IF eState = E_MethodKeepAliveMotionSystem.eIdle THEN
	MEMSET(ADR(stRtPartActivatePosition), 0, SIZEOF(stRtPartActivatePosition));
	stRtPartActivatePosition.Busy := TRUE;
	
	    nPartActivateIndex := nPartIndex;
	nPositionActivateIndex := nPositionIndex;
	  
	              eState := E_MethodKeepAliveMotionSystem.ePartActivatePosition;
	PartActivatePosition := TRUE;
ELSE
	PartActivatePosition := FALSE;
END_IF
END_METHOD

METHOD PartAllowEnable : BOOL
VAR_INPUT
	nPartID		: UDINT;
END_VAR


IF eState = E_MethodKeepAliveMotionSystem.eIdle THEN
	MEMSET(ADR(stRtPartAllowEnable), 0, SIZEOF(stRtPartAllowEnable));
	     PartToEnableAllow := nPartID;
	           eState := E_MethodKeepAliveMotionSystem.ePartAllowEnable;
	  PartAllowEnable := TRUE;
ELSE
	PartAllowEnable := FALSE;
END_IF
END_METHOD

METHOD PartForceDisable : BOOL
VAR_INPUT
	nPartID		: UDINT;
END_VAR


IF eState = E_MethodKeepAliveMotionSystem.eIdle THEN
	MEMSET(ADR(stRtPartForceDisable), 0, SIZEOF(stRtPartForceDisable));
	   PartToDisable := nPartID;
	          eState := E_MethodKeepAliveMotionSystem.ePartForceDisable;
	  PartForceDisable := TRUE;
ELSE
	PartForceDisable := FALSE;
END_IF
END_METHOD

METHOD PartForceEnable : BOOL
VAR_INPUT
	nPartID		: UDINT;
END_VAR


IF  eState  = E_MethodKeepAliveMotionSystem.eIdle
AND nPartID > 0 
THEN
		MEMSET(ADR(stRtPartForceEnable), 0, SIZEOF(stRtPartForceEnable));
		PartToEnableForce := nPartID;
				   eState := E_MethodKeepAliveMotionSystem.ePartForceEnable;
		  PartForceEnable := TRUE;
ELSE
	PartForceEnable := FALSE;
END_IF
END_METHOD

METHOD PartInitialize : BOOL
VAR_INPUT
	nPartID		: OTCID;
END_VAR



IF eState = E_MethodKeepAliveMotionSystem.eIdle THEN
	MEMSET(ADR(stRtPartInitialize), 0, SIZEOF(stRtPartInitialize));
	PartToInitialze := nPartID;
	       eState := E_MethodKeepAliveMotionSystem.ePartInitialize;
	  PartInitialize := TRUE;
ELSE
	PartInitialize := FALSE;
END_IF
END_METHOD

METHOD PartInitializeMulti : BOOL
VAR_INPUT
	
	AdrPartID		: PVOID;
	nPartCount		: UINT;
	
END_VAR

IF eState = E_MethodKeepAliveMotionSystem.eIdle THEN
	MEMSET(ADR(stRtPartInitializeMulti), 0, SIZEOF(stRtPartInitializeMulti));
	
	AddressArrayPartID	:= AdrPartID;
	          nPartCnt	:= nPartCount;		
	
	       eState := E_MethodKeepAliveMotionSystem.ePartInitializeMulti;
	  PartInitializeMulti := TRUE;
ELSE
	PartInitializeMulti := FALSE;
END_IF
END_METHOD

METHOD PartReset : BOOL
VAR_INPUT
	nPartID		: UDINT;
END_VAR


IF eState = E_MethodKeepAliveMotionSystem.eIdle THEN
	MEMSET(ADR(stRtPartReset), 0, SIZEOF(stRtPartReset));
	      PartToReset := nPartID;
	           eState := E_MethodKeepAliveMotionSystem.ePartReset;
	        PartReset := TRUE;
ELSE
	PartReset := FALSE;
END_IF
END_METHOD

METHOD RemoveEnvironmentFromGroup : BOOL
IF eState = E_MethodKeepAliveMotionSystem.eIdle THEN
	MEMSET(ADR(stRtRemoveEnvironment), 0, SIZEOF(stRtRemoveEnvironment));
	eState := E_MethodKeepAliveMotionSystem.eRemoveEnvironmentFromGroup;
	RemoveEnvironmentFromGroup := TRUE;
ELSE
	RemoveEnvironmentFromGroup := FALSE;
END_IF
END_METHOD

METHOD RemoveMoverFromGroup : BOOL
VAR_INPUT
	ipMover		: I_XPlanarMoverStandard;
END_VAR
IF eState = E_MethodKeepAliveMotionSystem.eIdle THEN
	MEMSET(ADR(stRtRemoveMover), 0, SIZEOF(stRtRemoveMover));
	eState := E_MethodKeepAliveMotionSystem.eRemoveMoverFromGroup;
	MoverToRemove := ipMover;
	RemoveMoverFromGroup := TRUE;
ELSE
	RemoveMoverFromGroup := FALSE;
END_IF
END_METHOD

METHOD RemoveMoversFromGroup : BOOL
IF eState = E_MethodKeepAliveMotionSystem.eIdle THEN
	MEMSET(ADR(stRtRemoveMovers), 0, SIZEOF(stRtRemoveMovers));
	eState := E_MethodKeepAliveMotionSystem.eRemoveMoversFromGroup;
	RemoveMoversFromGroup := TRUE;
ELSE
	RemoveMoversFromGroup := FALSE;
END_IF
END_METHOD

METHOD RemoveTracksFromGroup : BOOL



VAR_INST
	nTestCounter01 : UINT;	
	
END_VAR
IF eState = E_MethodKeepAliveMotionSystem.eIdle THEN
	MEMSET(ADR(stRtRemoveTracks), 0, SIZEOF(stRtRemoveTracks));
	eState := E_MethodKeepAliveMotionSystem.eRemoveTracksFromGroup;
	RemoveTracksFromGroup := TRUE;
	
	nTestCounter01 := nTestCounter01 +1;
ELSE
	RemoveTracksFromGroup := FALSE;
END_IF
END_METHOD

METHOD ResetGroup : BOOL
IF eState = E_MethodKeepAliveMotionSystem.eIdle THEN
	MEMSET(ADR(stRtResetGroup), 0, SIZEOF(stRtResetGroup));
	eState := E_MethodKeepAliveMotionSystem.eResetGroup;
	ResetGroup := TRUE;
ELSE
	ResetGroup := FALSE;
END_IF
END_METHOD

METHOD ResetMovers : BOOL
IF eState = E_MethodKeepAliveMotionSystem.eIdle THEN
	MEMSET(ADR(stRtResetMovers), 0, SIZEOF(stRtResetMovers));
	eState := E_MethodKeepAliveMotionSystem.eResetMovers;
	ResetMovers := TRUE;
ELSE
	ResetMovers := FALSE;
END_IF
END_METHOD

METHOD ResetParts : BOOL
IF eState = E_MethodKeepAliveMotionSystem.eIdle THEN
	MEMSET(ADR(stRtResetParts), 0, SIZEOF(stRtResetParts));
	eState := E_MethodKeepAliveMotionSystem.eResetParts;
	ResetParts := TRUE;
ELSE
	ResetParts := FALSE;
END_IF
END_METHOD

METHOD ResetTracks : BOOL
IF eState = E_MethodKeepAliveMotionSystem.eIdle THEN
	MEMSET(ADR(stRtResetTracks), 0, SIZEOF(stRtResetTracks));
	eState := E_MethodKeepAliveMotionSystem.eResetTracks;
	ResetTracks := TRUE;
ELSE
	ResetTracks := FALSE;
END_IF
END_METHOD

METHOD UtilityCheckForError : DINT
VAR_INPUT
	bAutoReset : BOOL;
END_VAR
	IF bAutoReset THEN
		IF ipXpuInternal.Error THEN
			ipXpuInternal.ErrorAcknowledge();
		END_IF
	END_IF

	IF ipXpuInternal.Error THEN
		UtilityCheckForError := -1;
	ELSE
		UtilityCheckForError := +1;
	END_IF
END_METHOD

METHOD UtilityErrorReset : BOOL
VAR_INPUT
END_VAR
IF ipXpuInternal.Error THEN
	ipXpuInternal.ErrorAcknowledge();
END_IF
END_METHOD

METHOD PROTECTED ccl_AddEnvironmentToGroup : BOOL

VAR
	EmptyOT : EPlanarObjectType;
END_VAR

CASE nState OF
	

	0:  // Prepare
		stRtAddEnvironment.Aborted := FALSE;
		stRtAddEnvironment.Active  := TRUE;
		stRtAddEnvironment.Done    := FALSE;
		stRtAddEnvironment.Busy    := TRUE;
		stRtAddEnvironment.Error   := FALSE;
		stRtAddEnvironment.ErrorID := 0;
		stRtAddEnvironment.stInfo  := _stResultErrorInfoClear;
		
		nState := 5;


	5:  // Checking if the environment already belongs to the group
		IF environment.MCTOPLC_STD.GroupOID = 0 THEN
			environment.CreateBoundary(cmdFeedback);
			nState := 10;
		ELSE
			nState := 110;
		END_IF
	
		
	10:	// Creating the boundary 
		environment.CreateBoundary(cmdFeedback);
		nState := nState + 1;
			
	11:	IF cmdFeedback.Done THEN
			nState := 20;
		ELSIF cmdFeedback.Error THEN
			nState := 100;
		END_IF
		
		
	20:	// Adding the environment to the group
		environment.AddToGroup(cmdFeedback, group);
		nState := nState + 1;

	21:	IF cmdFeedback.Done 
		OR cmdFeedback.Error
		THEN
			nState := 100;
		END_IF
		
		
		
	100: // Result with action
		stRtAddEnvironment.Aborted            := FALSE;
		stRtAddEnvironment.Active             := FALSE;
		stRtAddEnvironment.Busy               := FALSE;
		stRtAddEnvironment.Done               := cmdFeedback.Done;
		stRtAddEnvironment.Error              := cmdFeedback.Error;
		stRtAddEnvironment.ErrorID            := cmdFeedback.ErrorId;
		stRtAddEnvironment.stInfo.nObjectID   := cmdFeedback.objectInfo.Id;
		stRtAddEnvironment.stInfo.nObjectType := cmdFeedback.objectInfo.ObjectType;
		nState := 200;
		
		
	110: // Result without action
		stRtAddEnvironment.Aborted            := FALSE;
		stRtAddEnvironment.Active             := FALSE;
		stRtAddEnvironment.Busy               := FALSE;
		stRtAddEnvironment.Done               := TRUE;
		stRtAddEnvironment.Error              := FALSE;
		stRtAddEnvironment.ErrorID            := 0;
		stRtAddEnvironment.stInfo.nObjectID   := 0;
		stRtAddEnvironment.stInfo.nObjectType := EmptyOT;
		nState := 200;		
		
		
	200: // Done	
		eState := E_MethodKeepAliveMotionSystem.eIdle;
		nState := 0;		
		ccl_AddEnvironmentToGroup := TRUE;
		
		
END_CASE
END_METHOD

METHOD PROTECTED ccl_AddModuleToEnvironment : BOOL

CASE nState OF
	
	0: 	// Prepare
		stRtAddModule.Aborted := FALSE;
		stRtAddModule.Active  := TRUE;
		stRtAddModule.Busy	  := TRUE;
		stRtAddModule.Done 	  := FALSE;
		stRtAddModule.Error   := FALSE;
		stRtAddModule.ErrorID := 0;
		stRtAddModule.stInfo  := _stResultErrorInfoClear;
		nState := 10;
	
		
	10: // Adding the tile	
		environment.AddStator(cmdFeedback, _addModulePositionX, _addModulePositionY);
		nState := nState + 10;
		
		
	20: // Checking command feedback
		IF cmdFeedback.Done
		OR cmdFeedback.Error
		THEN
			                  _bResultDone  := cmdFeedback.Done;
			                  _bResultError := cmdFeedback.Error;
			                _nResultErrorID := cmdFeedback.ErrorId;
			   _stResultErrorInfo.nObjectID := cmdFeedback.objectInfo.Id;	
			 _stResultErrorInfo.nObjectType := cmdFeedback.objectInfo.ObjectType;	
			    		 nState := 100;
		END_IF		

		
	100:  // Done	
		stRtAddModule.Aborted	:= FALSE;
		stRtAddModule.Active	:= FALSE;
		stRtAddModule.Busy   	:= FALSE;
		stRtAddModule.Done   	:= _bResultDone;
		stRtAddModule.Error		:= _bResultError;
		stRtAddModule.ErrorID	:= _nResultErrorID;
		stRtAddModule.stInfo	:= _stResultErrorInfo;
		
		eState := E_MethodKeepAliveMotionSystem.eIdle;
		nState := 0;
		ccl_AddModuleToEnvironment := TRUE;	

END_CASE
END_METHOD

METHOD PROTECTED ccl_AddMoversToGroup : BOOL



CASE nState OF
	
	0:  // Prepare
		stRtAddMovers.Aborted := FALSE;
		stRtAddMovers.Active  := FALSE;
		stRtAddMovers.Busy    := TRUE;
		stRtAddMovers.Error   := FALSE;
		stRtAddMovers.ErrorID := 0;
		stRtAddMovers.stInfo  := _stResultErrorInfoClear;

		nState := 10;
	
	
	10: // Adding movers to the group
		stRtAddMovers.Active := TRUE;
		bDone := TRUE;
		FOR nForCounter := 1 TO _nAxisCount DO
			IF ipMover[nForCounter].P_PhysicalAreaID > 0 THEN
				bDone := bDone AND ipMover[nForCounter].AddToGroup(group);
			END_IF
		END_FOR
		IF bDone THEN
			nState := 20;
		END_IF
		
		
	20: // Checking command feedback
		_nResultErrorID    := 0;
		_stResultErrorInfo := _stResultErrorInfoClear;
	
		bError := FALSE;
		bDone  := TRUE;
		FOR nForCounter := 1 TO _nAxisCount DO
			IF ipMover[nForCounter].P_PhysicalAreaID > 0 THEN	
				bDone := bDone  AND ipMover[nForCounter].P_AddToGroup.Done;
				
				IF ipMover[nForCounter].P_AddToGroup.Error THEN
						bError := TRUE;
					   _nResultErrorID := ipMover[nForCounter].P_AddToGroup.ErrorID;
					_stResultErrorInfo := ipMover[nForCounter].P_AddToGroup.stInfo;
				END_IF
			END_IF
		END_FOR
		
		IF bDone 
		OR bError
		THEN
			_bResultDone  := bDone;
			_bResultError := bError;	
				   nState := 100;		
		END_IF
		
		
	100:  // Done
		stRtAddMovers.Aborted 	:= FALSE;
		stRtAddMovers.Active	:= FALSE;
		stRtAddMovers.Busy	    := FALSE;
		stRtAddMovers.Done      := _bResultDone;
		stRtAddMovers.Error     := _bResultError;
		stRtAddMovers.ErrorID	:= _nResultErrorID;
		stRtAddMovers.stInfo    := _stResultErrorInfo;
		
		eState := E_MethodKeepAliveMotionSystem.eIdle;
		nState := 0;
		ccl_AddMoversToGroup := TRUE;
		

END_CASE
END_METHOD

METHOD PROTECTED ccl_AddMoverToGroup : BOOL


VAR_INPUT
	ipMoverToAdd	: I_XPlanarMoverStandard;
END_VAR


VAR_INST
	nMoverToAdd		: UDINT;	
END_VAR


CASE nState OF

	0: // Prepare
		stRtAddMover.Aborted := FALSE;
		stRtAddMover.Active  := TRUE;
		stRtAddMover.Busy    := TRUE;
		stRtAddMover.Done    := FALSE;
		stRtAddMover.Error	 := FALSE;
		stRtAddMover.ErrorID := 0;
		stRtAddMover.stInfo	 := _stResultErrorInfoClear;
		
		nState := 10;
	
	10: // Adding the mover to the group
		      bDone := TRUE;		
		nMoverToAdd := 0;
		FOR idx:=1 TO Params_XPlanar.maxNumMover DO
			IF  ipMover[idx] <> 0			 
			AND ipMover[idx] = ipMoverToAdd
			THEN
				nMoverToAdd := idx;	
				EXIT;
			END_IF
		END_FOR
		
		IF nMoverToAdd > 0 THEN
			ipMover[nMoverToAdd].AddToGroup(group);
			nState := 20;	
		ELSE
			nState := 30;	
		END_IF
		

	20: // Checking feedback
		_bResultDone       := ipMover[nMoverToAdd].P_AddToGroup.Done;
		_bResultError      := ipMover[nMoverToAdd].P_AddToGroup.Error;
		_nResultErrorID    := ipMover[nMoverToAdd].P_AddToGroup.ErrorID;
		_stResultErrorInfo := ipMover[nMoverToAdd].P_AddToGroup.stInfo;
		
		IF _bResultDone
		OR _bResultError
		THEN
			nState := 100;
		END_IF
		
		
	30:	// Error - no mover to add = undefined error
		_bResultDone       := FALSE;
		_bResultError      := TRUE;
		_nResultErrorID    := 0;
		_stResultErrorInfo := _stResultErrorInfoClear;		
		            nState := 100;
	
		
	100: // Done	
		stRtAddMover.Active  := FALSE;		
		stRtAddMover.Busy    := FALSE;
		stRtAddMover.Done    := _bResultDone;		
		stRtAddMover.Error   := _bResultError;
		stRtAddMover.ErrorID := _nResultErrorID;
		stRtAddMover.stInfo  := _stResultErrorInfo; 			

		eState := E_MethodKeepAliveMotionSystem.eIdle;
		nState := 0;		
		ccl_AddMoverToGroup := TRUE;
		

END_CASE
END_METHOD

METHOD PROTECTED ccl_AddTracksToGroup : BOOL



VAR_INST
	
	nTestCounter01	: UINT;
	
END_VAR
CASE nState OF
	
	0:  // Prepare
		stRtAddTracks.Aborted  := FALSE;
		stRtAddTracks.Active   := TRUE;
		stRtAddTracks.Busy     := TRUE;
		stRtAddTracks.Done     := FALSE;
		stRtAddTracks.Error    := FALSE;
		stRtAddTracks.ErrorID  := 0;
		stRtAddTracks.stInfo   := _stResultErrorInfoClear;

		nState := 10;
		
		nTestCounter01 := nTestCounter01 +1;
	
		
	10: // Adding tracks to the group
		bDone := TRUE;
		FOR nForCounter := 1 TO _nTrackCount DO
			bDone := bDone AND ipTrack[nForCounter].AddToGroup(group);
		END_FOR
		
		IF bDone THEN
			nState := 20;
		END_IF
		
		
	20: // Checking feedback 
		nErrorID := 0;
		  bError := FALSE;
		   bDone := TRUE;
		   
		FOR nForCounter := 1 TO _nTrackCount DO
			 bDone := bDone  AND ipTrack[nForCounter].P_AddToGroup.Done;
		
			IF NOT bError AND ipTrack[nForCounter].P_AddToGroup.Error THEN
				           bError := TRUE;
				         nErrorID := ipTrack[nForCounter].P_AddToGroup.ErrorID;
				stResultErrorInfo := ipTrack[nForCounter].P_AddToGroup.stInfo;
			END_IF
		END_FOR
		
		IF bDone OR bError THEN
			      _bResultDone := bDone;
			     _bResultError := bError;
			   _nResultErrorID := nErrorID;
			_stResultErrorInfo := stResultErrorInfo;
			            nState := 100;
		END_IF
		
	
	100:  // Done
		stRtAddTracks.Active  := FALSE;
		stRtAddTracks.Busy    := FALSE;
		stRtAddTracks.Done    := _bResultDone;
		stRtAddTracks.Error   := _bResultError;
		stRtAddTracks.ErrorID := _nResultErrorID;
		stRtAddTracks.stInfo  := _stResultErrorInfo;
		
		eState := E_MethodKeepAliveMotionSystem.eIdle;
		nState := 0;			   
		ccl_AddTracksToGroup  := TRUE;

END_CASE
END_METHOD

METHOD ccl_CheckValidMovers : BOOL
VAR_INPUT
END_VAR



VAR_INST
	
	nState		 : UDINT;
	
	nHardwareOID				: UDINT;
	nModuleOID					: UDINT;
	nParameterOID				: UDINT;
	nSizeOfParameter			: UDINT;
	ParameterAddress			: PVOID;
	
	
	fbReadReq    : ADSREAD := ( NETID := '', PORT := 501, TMOUT := DEFAULT_ADS_TIMEOUT );
	bReadADS	 : BOOL;	
	bReadBusy	 : BOOL;
	bReadError	 : BOOL;
	nReaderrorID : UDINT;
	
	
	ModuleOIDs		: ARRAY[1..Param_TcIoXPlanarEnvironment.MaxXPlanarMoversPerXpu] OF OTCID;
	nMoverIdx		: UINT;
	
	
	//PROPERTY ipTcIoMover : ARRAY [1..Params_XPlanar.maxNumMover] OF I_TcIoXPlanarMover;
	
	Movers					: ARRAY [1..Params_XPlanar.maxNumMover] OF I_TcIoXPlanarMover;
	MoverPositionInfoAct	: MoverPositionInfo;
	
	
	nMoverValidCount		: UDINT;	
	bAllMoversValid			: BOOL;
	bMoverLost				: BOOL;

	
	fCurrentPositionX_01		: LREAL;
	fCurrentPositionX_02		: LREAL;
	fFeedbackCheckRegister		: ARRAY [0..10] OF LREAL;
	nFeedbackCheckIdx			: UINT;
	idx							: UINT;
	nMatchCount					: UINT;
	bFreezeDetect				: BOOL;
	
	
END_VAR


	CASE nState OF
		
	0:	
		stValidMoverCheckInfo.bDone            := FALSE;
		stValidMoverCheckInfo.bAllMoversValid  := FALSE;
		stValidMoverCheckInfo.bMoverLost       := FALSE;
		stValidMoverCheckInfo.nValidMoverCount := 0;
	
		       nMoverIdx := 0;
			  bMoverLost := FALSE;
		nMoverValidCount := 0;
		          nState := 10;
				  
	10:
		nMoverIdx := nMoverIdx +1;
		IF nMoverIdx <= Params_XPlanar.maxNumMover AND nMoverIdx <= ipXpuInternal.GetMoverCount() AND ipMover[nMoverIdx] <> 0 THEN
			nState := nState + 10;
		ELSE
			nMoverIdx := nMoverIdx -1;
			   nState := 30;
		END_IF
	
	20:		
		IF ipMover[nMoverIdx] <> 0 AND nMoverIdx <= ipXpuInternal.GetMoverCount() THEN
			MoverPositionInfoAct := ipXpuInternal.MoverTcIo(nMoverIdx).GetActualPositions();
			IF  MoverPositionInfoAct.MovementAreaOID  <> 0
			AND MoverPositionInfoAct.ActualPosition.z  < 6.0
			THEN
				nMoverValidCount := nMoverValidCount +1;
			END_IF
			nState := nState - 10;
		END_IF

	30:
		IF nMoverValidCount = nMoverIdx THEN 
			bAllMoversValid := TRUE;
			nState := nState + 10; 
		ELSE
			bMoverLost := TRUE;
			nState := 100;
		END_IF
		
				
		
	40: // Check Feedback
		  nMoverIdx := 0;
		nMatchCount := 0;
		nState := nState + 1; 
		
	41:
		nMoverIdx := nMoverIdx +1;
		IF nMoverIdx <= Params_XPlanar.maxNumMover AND nMoverIdx <= ipXpuInternal.GetMoverCount() AND ipMover[nMoverIdx] <> 0 THEN
			nState := nState + 1; 
		ELSE
			nState := 100;
		END_IF
	

	42:
		MoverPositionInfoAct := ipXpuInternal.MoverTcIo(nMoverIdx).GetActualPositions();		
		fCurrentPositionX_01 := MoverPositionInfoAct.ActualPosition.x; 
		nState := nState + 1; 
		
	43:
		MoverPositionInfoAct := ipXpuInternal.MoverTcIo(nMoverIdx).GetActualPositions();		
		fCurrentPositionX_02 := MoverPositionInfoAct.ActualPosition.x;
		
		IF fCurrentPositionX_01 = fCurrentPositionX_02 THEN
			nMatchCount := nMatchCount +1;
			
			IF nMatchCount >= 4 THEN
				bFreezeDetect := TRUE;
				nState := nState + 1; 
			ELSE
				nState := nState - 1; 
			END_IF
		ELSE
			bFreezeDetect := FALSE;
			nState := nState + 1; 
		END_IF
		
	44:
		IF bFreezeDetect THEN
			bAllMoversValid := FALSE;
			     bMoverLost := TRUE;
	       nMoverValidCount := 0;
				 
			nState := 100;
		ELSE
			nState := 41;
		END_IF


		
		
	
	100:		
		stValidMoverCheckInfo.bAllMoversValid 	:= bAllMoversValid;
		stValidMoverCheckInfo.bMoverLost 		:= bMoverLost; 
		stValidMoverCheckInfo.bDone 			:= TRUE;
		stValidMoverCheckInfo.nValidMoverCount  := nMoverValidCount;
	
		eState := E_MethodKeepAliveMotionSystem.eIdle;
		nState := 0;
		
		
	
	END_CASE
END_METHOD

METHOD PROTECTED ccl_DisableGroup : BOOL

CASE nState OF 


	0:  // Prepare 
		stRtDisableGroup.Aborted  := FALSE;
		stRtDisableGroup.Active   := TRUE;
		stRtDisableGroup.Busy     := TRUE;
		stRtDisableGroup.Done     := FALSE;
		stRtDisableGroup.Error    := FALSE;
		stRtDisableGroup.ErrorID  := 0;
		stRtDisableGroup.stInfo   := _stResultErrorInfoClear;
	
		nState := 10;


	10: // Disabeling the group
		Group.Disable(CmdFeedback);
		nState := 20; 
		
		
	20: // Checking feedback
		                  _bResultDone := CmdFeedback.Done;
		                 _bResultError := CmdFeedback.Error;
		               _nResultErrorID := CmdFeedback.ErrorId;
		  _stResultErrorInfo.nObjectID := CmdFeedback.objectInfo.Id;   
		_stResultErrorInfo.nObjectType := CmdFeedback.objectInfo.ObjectType;
	
		IF _bResultDone
		OR _bResultError
		THEN
			nState := 100;	
		END_IF
	
		
	100:  // Done
		stRtDisableGroup.Aborted := FALSE;
		stRtDisableGroup.Active  := FALSE;
		stRtDisableGroup.Busy    := FALSE;
		stRtDisableGroup.Done    := _bResultDone;
		stRtDisableGroup.Error	 := _bResultError;
		stRtDisableGroup.ErrorID := _nResultErrorID;
		stRtDisableGroup.stInfo  := _stResultErrorInfo;
	
		eState := E_MethodKeepAliveMotionSystem.eIdle;
		nState := 0;	
		ccl_DisableGroup := TRUE;
			
END_CASE
END_METHOD

METHOD PROTECTED ccl_DisableMovers : BOOL



CASE nState OF
	

	0:  // Prepare
		stRtDisableMovers.Aborted  := FALSE;
		stRtDisableMovers.Active   := TRUE;
		stRtDisableMovers.Busy     := TRUE;
		stRtDisableMovers.Done	   := FALSE;
		stRtDisableMovers.Error    := FALSE;
		stRtDisableMovers.ErrorID  := 0;
		stRtDisableMovers.stInfo   := _stResultErrorInfoClear;
	
		nErrorID := 0;
		nState:= 10;
	
		
	10: // Disable all movers
		FOR nForCounter := 1 TO _nAxisCount DO
			IF ipMover[nForCounter].P_PhysicalAreaID > 0 THEN
				ipMover[nForCounter].Disable('Disable all Movers');
			END_IF
		END_FOR
		nState := 20;
		
		
	20:  // Checking feedback
		 bDone := TRUE;
		bError := FALSE;
		FOR nForCounter := 1 TO _nAxisCount DO
			IF ipMover[nForCounter].P_PhysicalAreaID > 0 THEN
				bDone := bDone AND ipMover[nForCounter].P_Disable.Done;
				
				IF NOT bError AND ipMover[nForCounter].P_Disable.Error THEN
							   bError := TRUE;
							 nErrorID := ipMover[nForCounter].P_Disable.ErrorID;
					stResultErrorInfo := ipMover[nForCounter].P_Disable.stInfo;
				END_IF
			END_IF
		END_FOR	
			
		IF bDone OR bError THEN
			nState := 21;
		END_IF

	21:
		_bResultDone 		:= bDone;
		_bResultError 		:= bError;
		_nResultErrorID		:= nErrorID;
		_stResultErrorInfo	:= stResultErrorInfo;
		nState := 100;
		
	
	100:  // Done
		stRtDisableMovers.Aborted  := FALSE;
		stRtDisableMovers.Active   := FALSE;
		stRtDisableMovers.Busy     := FALSE;
		stRtDisableMovers.Done	   := _bResultDone;
		stRtDisableMovers.Error    := _bResultError;
		stRtDisableMovers.ErrorID  := _nResultErrorID;
		stRtDisableMovers.stInfo   := _stResultErrorInfo;		
	
		eState := E_MethodKeepAliveMotionSystem.eIdle;
		nState := 0;
		ccl_DisableMovers := TRUE;
		
END_CASE
END_METHOD

METHOD PROTECTED ccl_DisableTracks : BOOL

VAR_INST

	nTrackToDisable		: INT;
	nTrackToDisableCNT	: INT;
		
	nTestCounter01		: UINT;
	nTestCounter02		: UINT;
	nLastTrackDisabled 	: INT;
	
END_VAR
CASE nState OF
	

	0:  // Prepare
		stRtDisableTracks.Aborted  := FALSE;
		stRtDisableTracks.Active   := TRUE;
		stRtDisableTracks.Busy     := TRUE;
		stRtDisableTracks.Done     := FALSE; 
		stRtDisableTracks.Error    := FALSE; 
		stRtDisableTracks.ErrorID  := 0;
		stRtDisableTracks.stInfo   := _stResultErrorInfoClear;
	
		nState := 10;
		
		nTestCounter01 := nTestCounter01 +1;
		
		
	10:  // Disabeling all tracks one-by-one
			     nTestCounter02 := nTestCounter02 +1;
				 
				 		  bError := FALSE;
				           bDone := FALSE;
		         nTrackToDisable := 0;
		      nTrackToDisableCNT := 0;
	          nLastTrackDisabled := 0;
		stRtEnableTracks.Active := TRUE;
		                 nState := 11;
		
	11:	// Checking if track is real
		nTrackToDisableCNT := nTrackToDisableCNT +1;
		IF nTrackToDisableCNT <= _nTrackCount THEN
			IF ipTrack[nTrackToDisableCNT] <> 0 THEN
				   nTrackToDisable := nTrackToDisableCNT;
				nLastTrackDisabled := nTrackToDisable;
				nState := nState +1;
			ELSE
				nState := 20;
			END_IF
		ELSE
			 bDone := TRUE;
			nState := 20;
		END_IF
		
		
	12:	// Disabeling
		IF ipTrack[nTrackToDisable].Disable() THEN
			nState := nState +1;
		END_IF
	
			
	13:	// Checking feedback
		IF ipTrack[nTrackToDisable].P_Disable.Done THEN
			nState := nState -2;
		ELSIF ipTrack[nTrackToDisable].P_Disable.Error THEN
				         bError := ipTrack[nTrackToDisable].P_Disable.Error;
				       nErrorID := ipTrack[nTrackToDisable].P_Disable.ErrorID;
			  stResultErrorInfo := ipTrack[nTrackToDisable].P_Disable.stInfo;
		
			nState := 20;
		END_IF
			
	
	20:	// All tracks are through
				  _bResultDone := bDone;
				 _bResultError := bError;
			   _nResultErrorID := nErrorID;
			_stResultErrorInfo := stResultErrorInfo;		

			nState := 100;				
	
	
	100:  // Done	
		stRtDisableTracks.Active   := FALSE;
		stRtDisableTracks.Busy     := FALSE;
		stRtDisableTracks.Done 	   := _bResultDone;
		stRtDisableTracks.Error    := _bResultError;
		stRtDisableTracks.ErrorID  := _nResultErrorID;
		stRtDisableTracks.stInfo   := _stResultErrorInfo;
		
		           eState := E_MethodKeepAliveMotionSystem.eIdle;
				   nState := 0;
		ccl_DisableTracks := TRUE;
		
			
END_CASE
END_METHOD

METHOD PROTECTED ccl_EnableGroup : BOOL




CASE nState OF 
	
	0:  // Prepare
		stRtEnableGroup.Aborted  := FALSE;
		stRtEnableGroup.Active   := TRUE;
		stRtEnableGroup.Busy     := TRUE;
		stRtEnableGroup.Done     := FALSE;
		stRtEnableGroup.Error    := FALSE;
		stRtEnableGroup.ErrorID  := 0;
		stRtEnableGroup.stInfo   := _stResultErrorInfoClear;
	
		nState := 10;
	
	
	10: // Activating the group
		group.Enable(cmdFeedback);
		nState := 11;
	
	
	11: // Checking feedback
		                  _bResultDone := cmdFeedback.Done;
		                 _bResultError := cmdFeedback.Error;
		               _nResultErrorID := cmdFeedback.ErrorId;
		  _stResultErrorInfo.nObjectID := cmdFeedback.objectInfo.Id;
		_stResultErrorInfo.nObjectType := cmdFeedback.objectInfo.ObjectType;
	
		IF _bResultDone OR _bResultError THEN
			nState := 100;
		END_IF
	
		
	100:  // Done
		stRtEnableGroup.Aborted  := FALSE;
		stRtEnableGroup.Active   := FALSE;
		stRtEnableGroup.Busy     := FALSE;
		stRtEnableGroup.Done     := _bResultDone;
		stRtEnableGroup.Error    := _bResultError;
		stRtEnableGroup.ErrorID  := _nResultErrorID;
		stRtEnableGroup.stInfo   := _stResultErrorInfo;	
	
		eState := E_MethodKeepAliveMotionSystem.eIdle;
		nState := 0;
		ccl_EnableGroup := TRUE;
	
		
END_CASE
END_METHOD

METHOD PROTECTED ccl_EnableMovers : BOOL


CASE nState OF

	0:	// Prepare 
		stRtEnableMovers.Aborted  := FALSE;
		stRtEnableMovers.Active   := TRUE;
		stRtEnableMovers.Busy	  := TRUE;
		stRtEnableMovers.Done     := FALSE;
		stRtEnableMovers.Error    := FALSE;
		stRtEnableMovers.ErrorID  := 0;
		stRtEnableMovers.stInfo	  := _stResultErrorInfoClear;

		nState := 10;
		
		
	10:  // Enabeling all movers
		bDone := TRUE;
		FOR nForCounter := 1 TO _nAxisCount DO
			IF ipMover[nForCounter].P_PhysicalAreaID > 0 THEN
				bDone := bDone AND ipMover[nForCounter].Enable('Enable all Movers');
			END_IF
		END_FOR
		IF bDone THEN
			nState := 20;
		END_IF
		
	20:  // Checking feedback
		 bDone := TRUE;
		bError := FALSE;
		FOR nForCounter := 1 TO _nAxisCount DO
			IF ipMover[nForCounter].P_PhysicalAreaID > 0 THEN
				bDone := bDone AND ipMover[nForCounter].P_Enable.Done;
			
				IF NOT bError AND ipMover[nForCounter].P_Enable.Error THEN
							   bError := TRUE;
							 nErrorID := ipMover[nForCounter].P_Enable.ErrorID;
					stResultErrorInfo := ipMover[nForCounter].P_Enable.stInfo;
				END_IF	
			END_IF
		END_FOR	
		
		IF bDone OR bError THEN
				  _bResultDone := bDone;
				 _bResultError := bError;
			   _nResultErrorID := nErrorID;
			_stResultErrorInfo := stResultErrorInfo;			
		
			nState := 100;
		END_IF
		
			
	100:  // Done
		stRtEnableMovers.Aborted  := FALSE;
		stRtEnableMovers.Active   := FALSE;
		stRtEnableMovers.Busy	  := FALSE;
		stRtEnableMovers.Done     := _bResultDone;
		stRtEnableMovers.Error    := _bResultError;
		stRtEnableMovers.ErrorID  := _nResultErrorID;
		stRtEnableMovers.stInfo	  := _stResultErrorInfo;
	
		eState := E_MethodKeepAliveMotionSystem.eIdle;
		nState := 0;
		ccl_EnableMovers := TRUE;
			

	
END_CASE
END_METHOD

METHOD PROTECTED ccl_EnableTrack : BOOL

VAR_INPUT
	ipTrackToEnable	: I_TrackStandard;
END_VAR






CASE nState OF

	0:  // Prepare
		stRtEnableTrack.Aborted := FALSE;
		stRtEnableTrack.Active  := TRUE;
		stRtEnableTrack.Busy    := TRUE;
		stRtEnableTrack.Done    := FALSE;
		stRtEnableTrack.Error   := FALSE;
		stRtEnableTrack.ErrorID := 0;
		stRtEnableTrack.stInfo  := _stResultErrorInfoClear;

		nState := 10;
		
		
	10: // Enable the track
		IF ipTrackToEnable.Enable() THEN
			nState := 20;
		END_IF
	
	
	20: // Checking feedback
		 _bResultDone := ipTrackToEnable.P_Enable.Done;
		_bResultError := ipTrackToEnable.P_Enable.Error;		
	
		IF _bResultDone OR _bResultError THEN
			        _nResultErrorID := ipTrackToEnable.P_Enable.ErrorID;
			     _stResultErrorInfo := ipTrackToEnable.P_Enable.stInfo;
			nState := 100;
		END_IF
		

	100: // Done
		stRtEnableTrack.Aborted := FALSE;
		stRtEnableTrack.Active  := FALSE;
		stRtEnableTrack.Busy    := FALSE;
		stRtEnableTrack.Done    := _bResultDone;
		stRtEnableTrack.Error   := _bResultError;
		stRtEnableTrack.ErrorID := _nResultErrorID;
		stRtEnableTrack.stInfo  := _stResultErrorInfo;

		         eState := E_MethodKeepAliveMotionSystem.eIdle;
				 nState := 0;
		ccl_EnableTrack := TRUE;
		
				
END_CASE
END_METHOD

METHOD PROTECTED ccl_EnableTracks : BOOL

VAR_INST

	nTrackToEnable		: INT;
	nTrackToEnableCNT	: INT;
		
	nTestCounter01		: UINT;
	nTestCounter02		: UINT;
	nLastTrackEnabled 	: INT;
	
END_VAR
CASE nState OF
	

	0:  // Prepare
		stRtEnableTracks.Aborted  := FALSE;
		stRtEnableTracks.Active   := TRUE;
		stRtEnableTracks.Busy     := TRUE;
		stRtEnableTracks.Done     := FALSE; 
		stRtEnableTracks.Error    := FALSE; 
		stRtEnableTracks.ErrorID  := 0;
		stRtEnableTracks.stInfo   := _stResultErrorInfoClear;
	
		nState := 10;
		
		nTestCounter01 := nTestCounter01 +1;
		
		
	10:  // Enabeling all tracks one-by-one
			     nTestCounter02 := nTestCounter02 +1;
				 
				 		 bError := FALSE;
				          bDone := FALSE;
		         nTrackToEnable := 0;
		      nTrackToEnableCNT := 0;
	          nLastTrackEnabled := 0;
		stRtEnableTracks.Active := TRUE;
		                 nState := 11;
		
	11:	// Checking if track is real
		nTrackToEnableCNT := nTrackToEnableCNT +1;
		IF nTrackToEnableCNT <= _nTrackCount THEN
			IF ipTrack[nTrackToEnableCNT] <> 0 THEN
				IF ipTrack[nTrackToEnableCNT].GetLength() > 0 THEN
					   nTrackToEnable := nTrackToEnableCNT;
					nLastTrackEnabled := nTrackToEnable;
					nState := nState +1;
				END_IF
			END_IF
		ELSE
			 bDone := TRUE;
			nState := 20;
		END_IF
		
		
	12:	// Enabeling
		IF ipTrack[nTrackToEnable].Enable() THEN
			nState := nState +1;
		END_IF
	
			
	13:	// Checking feedback
		IF ipTrack[nTrackToEnable].P_Enable.Done THEN
			nState := nState -2;
		ELSIF ipTrack[nTrackToEnable].P_Enable.Error THEN
				         bError := ipTrack[nTrackToEnable].P_Enable.Error;
				       nErrorID := ipTrack[nTrackToEnable].P_Enable.ErrorID;
			  stResultErrorInfo := ipTrack[nTrackToEnable].P_Enable.stInfo;
		
			nState := 20;
		END_IF
			
	
	20:	// All tracks are through
				  _bResultDone := bDone;
				 _bResultError := bError;
			   _nResultErrorID := nErrorID;
			_stResultErrorInfo := stResultErrorInfo;		

			nState := 100;				
	
	
	100:  // Done	
		stRtEnableTracks.Active   := FALSE;
		stRtEnableTracks.Busy     := FALSE;
		stRtEnableTracks.Done 	  := _bResultDone;
		stRtEnableTracks.Error 	  := _bResultError;
		stRtEnableTracks.ErrorID  := _nResultErrorID;
		stRtEnableTracks.stInfo   := _stResultErrorInfo;
		
		          eState := E_MethodKeepAliveMotionSystem.eIdle;
				  nState := 0;
		ccl_EnableTracks := TRUE;
		
			
END_CASE
END_METHOD

METHOD PROTECTED ccl_HaltSystem : BOOL

CASE nState OF
	
	0:  // Prepare 
		stRtHaltSystem.Aborted := FALSE;
		stRtHaltSystem.Active  := TRUE;
		stRtHaltSystem.Busy    := TRUE;
		stRtHaltSystem.Done    := FALSE;
		stRtHaltSystem.Error   := FALSE;
		stRtHaltSystem.ErrorID := 0;
		stRtHaltSystem.stInfo  := _stResultErrorInfoClear;

		nState := 10;
	
		
	10: // Halt to all moving movers
		bDone := TRUE;
		FOR nForCounter := 1 TO _nAxisCount DO
			IF ipMover[nForCounter] <> 0 THEN
				IF ipMover[nForCounter].P_Busy THEN
					bDone := bDone AND ipMover[nForCounter].Halt('HaltSystem');
				ELSE
					bDone := bDone AND TRUE;
				END_IF
			END_IF 
		END_FOR
		IF bDone THEN
			nState := 20;
		END_IF
		
		
	20:  // Checking feedback
		bError := FALSE;
		  bDone:= TRUE;
		FOR nForCounter := 1 TO _nAxisCount DO
			IF ipMover[nForCounter] <> 0 THEN
				
				bDone := bDone AND (ipMover[nForCounter].P_Halt.Done OR NOT ipMover[nForCounter].P_Busy);
				
				IF NOT bError AND ipMover[nForCounter].P_Halt.Error THEN
					IF ipMover[nForCounter].P_Busy THEN	
						         nErrorID := ipMover[nForCounter].P_Halt.ErrorID;
						stResultErrorInfo := ipMover[nForCounter].P_Halt.stInfo;
						           bError := TRUE;
					END_IF 
				END_IF
				
			END_IF 
		END_FOR
		
		IF bDone OR bError THEN
				  _bResultDone := bDone;
				 _bResultError := bError;
			   _nResultErrorID := nErrorID;
			_stResultErrorInfo := stResultErrorInfo;					
		
			nState := 100;
		END_IF
		
		
	100:  // Done
		stRtHaltSystem.Aborted := FALSE;
		stRtHaltSystem.Active  := FALSE;
		stRtHaltSystem.Busy    := FALSE;
		stRtHaltSystem.Done    := _bResultDone;
		stRtHaltSystem.Error   := _bResultError;
		stRtHaltSystem.ErrorID := _nResultErrorID;
		stRtHaltSystem.stInfo  := _stResultErrorInfo;
	
		eState := E_MethodKeepAliveMotionSystem.eIdle;
		nState := 0;
		ccl_HaltSystem := TRUE;
		

	
END_CASE
END_METHOD

METHOD PROTECTED ccl_LeaveTrack : BOOL

VAR_INST
	ActPosition		: PositionXYC;
	stOptions 		: ST_LeaveTrackOptions;

END_VAR


CASE nState OF
	
	0:  // Prepare
		stRtLeaveTrack.Aborted  := FALSE;
		stRtLeaveTrack.Active   := TRUE;
		stRtLeaveTrack.Busy     := TRUE;
		stRtLeaveTrack.Done     := FALSE;
		stRtLeaveTrack.Error    := FALSE;
		stRtLeaveTrack.ErrorID  := 0;
		stRtLeaveTrack.stInfo	:= _stResultErrorInfoClear;

		nState := 10;
		
		
	10:  // All movers leave track
		bDone := TRUE;
		FOR nForCounter := 1 TO _nAxisCount DO
			IF ipMover[nForCounter] <> 0 THEN
				IF ipMover[nForCounter].P_CommandMode = MC_PLANAR_MOVER_COMMAND_MODE.OnTrack
				OR ipMover[nForCounter].P_CommandMode = MC_PLANAR_MOVER_COMMAND_MODE.JoiningTrack
				OR ipMover[nForCounter].P_SetOnTrack.TrackOID <> 0
				THEN
					ActPosition.SetValuesXYC(ipMover[nForCounter].P_SetPosition.x,ipMover[nForCounter].P_SetPosition.y,ipMover[nForCounter].P_SetPosition.c);
					stOptions.useOrientation := TRUE;
					ipMover[nForCounter].LeaveTrack('SystemLeaveTrack', ActPosition,100,1000,1000,10000,stOptions);
				END_IF
			END_IF
		END_FOR
		nState := 20;
		
		
	20:  // Checking feedback
		bError := FALSE;
		 bDone := TRUE;
		FOR nForCounter := 1 TO _nAxisCount DO
			IF ipMover[nForCounter].P_CommandMode = MC_PLANAR_MOVER_COMMAND_MODE.OnTrack
			OR ipMover[nForCounter].P_CommandMode = MC_PLANAR_MOVER_COMMAND_MODE.JoiningTrack
			OR ipMover[nForCounter].P_CommandMode = MC_PLANAR_MOVER_COMMAND_MODE.LeavingTrack
			OR ipMover[nForCounter].P_SetOnTrack.TrackOID <> 0
			THEN
				bDone := FALSE;
				
				IF ipMover[nForCounter].P_LeaveTrack.Error THEN
					IF NOT bError THEN
						           bError := TRUE;
						         nErrorID := ipMover[nForCounter].P_LeaveTrack.ErrorID;
						stResultErrorInfo := ipMover[nForCounter].P_LeaveTrack.stInfo;
					END_IF
				END_IF
			END_IF
		END_FOR	
	
		
		IF bDone OR bError THEN
				  _bResultDone := bDone;
				 _bResultError := bError;
			   _nResultErrorID := nErrorID;
			_stResultErrorInfo := stResultErrorInfo;				
		
			nState := 100;
		END_IF
	
	
	100:  // Done
		stRtLeaveTrack.Aborted  := FALSE;
		stRtLeaveTrack.Active   := FALSE;
		stRtLeaveTrack.Busy     := FALSE;
		stRtLeaveTrack.Done     := _bResultDone;
		stRtLeaveTrack.Error    := _bResultError;
		stRtLeaveTrack.ErrorID  := _nResultErrorID;
		stRtLeaveTrack.stInfo	:= _stResultErrorInfo;

		eState := E_MethodKeepAliveMotionSystem.eIdle;
		nState := 0;
		ccl_LeaveTrack := TRUE;	


END_CASE
END_METHOD

METHOD PROTECTED ccl_MethodKeepAlive : BOOL
VAR_INPUT
END_VAR




VAR_INST

	nTestCounter01	: UINT;
	nTestCounter02	: UINT;
	nTestCounter03	: UINT;
	nTestCounter04	: UINT;
	nTestCounter05	: UINT;
	nTestCounter06	: UINT;
	nTestCounter07	: UINT;
	nTestCounter08	: UINT;
	nTestCounter09	: UINT;
	nTestCounter10	: UINT;
	nTestCounter11	: UINT;
	nTestCounter12	: UINT;
	nTestCounter13	: UINT;
	nTestCounter14	: UINT;
	nTestCounter15	: UINT;
	nTestCounter16	: UINT;
	nTestCounter17	: UINT;
	nTestCounter18	: UINT;
	nTestCounter19	: UINT;
	nTestCounter20	: UINT;
	nTestCounter21	: UINT;
	nTestCounter22	: UINT;
	nTestCounter23	: UINT;
	nTestCounter24	: UINT;
	nTestCounter25	: UINT;
	nTestCounter26	: UINT;
	nTestCounter27	: UINT;
	nTestCounter28	: UINT;
	nTestCounter29	: UINT;
	nTestCounter30	: UINT;









END_VAR
CASE eState OF
	
	E_MethodKeepAliveMotionSystem.eIdle:
		nTestCounter01 := nTestCounter01 +1;
		nState := 0;
	
	E_MethodKeepAliveMotionSystem.eAddEnvironmentToGroup:
		nTestCounter02 := nTestCounter02 +1;
		ccl_AddEnvironmentToGroup();	
		
	E_MethodKeepAliveMotionSystem.eAddMoverToGroup:
		nTestCounter03 := nTestCounter03 +1;
		ccl_AddMoverToGroup(MoverToAdd);		
		
	E_MethodKeepAliveMotionSystem.eAddMoversToGroup:
		nTestCounter04 := nTestCounter04 +1;
		ccl_AddMoversToGroup();
		
	E_MethodKeepAliveMotionSystem.eDisableGroup:
		nTestCounter05 := nTestCounter05 +1;
		ccl_DisableGroup();
		
	E_MethodKeepAliveMotionSystem.eDisableMovers:
		nTestCounter06 := nTestCounter06 +1;
		ccl_DisableMovers();	
		
	//E_MethodKeepAliveMotionSystem.eDisableSystem:
	// 	nTestCounter07 := nTestCounter07 +1;
	//	ccl_DisableSystem();
		
	E_MethodKeepAliveMotionSystem.eEnableGroup:
		nTestCounter08 := nTestCounter08 +1;
		ccl_EnableGroup();
		
	E_MethodKeepAliveMotionSystem.eEnableMovers:
		nTestCounter09 := nTestCounter09 +1;
		ccl_EnableMovers();
		
	//E_MethodKeepAliveMotionSystem.eEnableSystem:
		nTestCounter10 := nTestCounter10 +1;
	//	ccl_EnableSystem();
		
	E_MethodKeepAliveMotionSystem.eHaltSystem:
		nTestCounter11 := nTestCounter11 +1;
		ccl_HaltSystem();
		
	E_MethodKeepAliveMotionSystem.eLeaveTrack:
		nTestCounter12 := nTestCounter12 +1;
		ccl_LeaveTrack();
	
	E_MethodKeepAliveMotionSystem.eRemoveMoverFromGroup:
		nTestCounter13 := nTestCounter13 +1;
		ccl_RemoveMoverFromGroup(MoverToRemove);

	E_MethodKeepAliveMotionSystem.eRemoveMoversFromGroup:
		nTestCounter14 := nTestCounter14 +1;
		ccl_RemoveMoversFromGroup();
	
	E_MethodKeepAliveMotionSystem.eRemoveEnvironmentFromGroup:
		nTestCounter15 := nTestCounter15 +1;
		ccl_RemoveEnvironmentFromGroup();	

	E_MethodKeepAliveMotionSystem.eRemoveTracksFromGroup:
		ccl_RemoveTracksFromGroup();		
			
	E_MethodKeepAliveMotionSystem.eResetGroup:
		nTestCounter16 := nTestCounter16 +1;
		ccl_ResetGroup();
		
	E_MethodKeepAliveMotionSystem.eResetMovers:
		nTestCounter17 := nTestCounter17 +1;
		ccl_ResetMovers();
		
	E_MethodKeepAliveMotionSystem.eResetTracks:
		nTestCounter18 := nTestCounter18 +1;
		ccl_ResetTracks();		
		
		
	//E_MethodKeepAliveMotionSystem.eResetSystem:
	//  nTestCounter19 := nTestCounter19 +1;
	//	ccl_ResetSystem();
		
	E_MethodKeepAliveMotionSystem.eAddTracksToGroup:
		nTestCounter20 := nTestCounter20 +1;
		ccl_AddTracksToGroup();

	E_MethodKeepAliveMotionSystem.eEnableTrack:
		nTestCounter21 := nTestCounter21 +1;
		ccl_EnableTrack(TrackToEnable);	
	
	E_MethodKeepAliveMotionSystem.eEnableTracks:
		nTestCounter22 := nTestCounter22 +1;
		ccl_EnableTracks();	
		
	E_MethodKeepAliveMotionSystem.eDisableTracks:
		ccl_DisableTracks();			
		
	E_MethodKeepAliveMotionSystem.eAddModuleToEnvironment:
		nTestCounter23 := nTestCounter23 +1;
		ccl_AddModuleToEnvironment();		
		
	E_MethodKeepAliveMotionSystem.eError:
		nTestCounter24 := nTestCounter24 +1;
		
	E_MethodKeepAliveMotionSystem.eCheckValidMovers:		
		ccl_CheckValidMovers();

	E_MethodKeepAliveMotionSystem.ePartInitialize:		
		ccl_PartInitialize();		
		
	E_MethodKeepAliveMotionSystem.ePartInitializeMulti:		
		ccl_PartInitializeMulti();		

	E_MethodKeepAliveMotionSystem.ePartActivatePosition:		
		ccl_PartActivatePosition();			

	E_MethodKeepAliveMotionSystem.ePartAllowEnable:		
		ccl_PartAllowEnable();	

	E_MethodKeepAliveMotionSystem.ePartForceEnable:		
		ccl_PartForceEnable();					
		
	E_MethodKeepAliveMotionSystem.ePartForceDisable:
		ccl_PartForceDisable();	
	
	E_MethodKeepAliveMotionSystem.ePartReset:
		ccl_PartReset();	
		
	E_MethodKeepAliveMotionSystem.eResetParts:
		ccl_ResetParts();			
		
END_CASE


IF eState <> E_MethodKeepAliveMotionSystem.eIdle THEN
	cmdFeedback.Update();
END_IF
END_METHOD

METHOD ccl_PartActivatePosition : BOOL

VAR_INST
	

	nState			: INT;
	
	feedback		: MC_PlanarFeedback;
	stInfo			: ST_CommandReturnInfo;
	nErrorSituation	: UDINT;
	

END_VAR



	CASE nState OF
		
	
	0: 
		stRtPartActivatePosition.Aborted := FALSE;
		stRtPartActivatePosition.Active  := FALSE;
		stRtPartActivatePosition.Busy    := TRUE;
		stRtPartActivatePosition.Error   := FALSE;
		stRtPartActivatePosition.ErrorID := 0;
		stRtPartActivatePosition.stInfo  := _stResultErrorInfoClear;
	

		part[nPartActivateIndex].ActivatePosition(feedback,nPositionActivateIndex);
		nState := nState +10;
		
		
	10:
		IF NOT feedback.Busy THEN
			nState := 100;
		END_IF 	
		
	
	100:  	
		stRtPartActivatePosition.Aborted := feedback.Aborted;
		stRtPartActivatePosition.Active  := feedback.Active;
		stRtPartActivatePosition.Busy    := feedback.Busy;
		stRtPartActivatePosition.Done    := feedback.Done;
		stRtPartActivatePosition.Error   := feedback.Error;
		stRtPartActivatePosition.ErrorID := feedback.ErrorId;
		stRtPartActivatePosition.stInfo  := stInfo;
		

		eState := E_MethodKeepAliveMotionSystem.eIdle;
		nState := 0;
		ccl_PartActivatePosition := TRUE;
			
	END_CASE

	feedback.Update();
END_METHOD

METHOD ccl_PartAllowEnable : BOOL

VAR_INST
	
	nState			: INT;
	nPartIDint		: UDINT;
	feedback		: MC_PlanarFeedback;
	stInfo			: ST_CommandReturnInfo;

END_VAR


	CASE nState OF
	
	0:
		part[PartToEnableAllow].AllowEnable(feedback);
		
		stRtPartAllowEnable.Active  := FALSE;
		stRtPartAllowEnable.Busy    := FALSE;
		
		nState	:= 10;
		
		
	10:
		IF feedback.Done
		OR feedback.Error
		THEN
			nState := 100;
		END_IF
			
		
	100:  // Done or Error
		stInfo.nObjectID := feedback.objectInfo.Id;
		stInfo.nObjectType := feedback.objectInfo.ObjectType;
	
	
		stRtPartAllowEnable.Aborted := FALSE;
		stRtPartAllowEnable.Active  := FALSE;
		stRtPartAllowEnable.Busy    := FALSE;
		stRtPartAllowEnable.Done    := feedback.Done;
		stRtPartAllowEnable.Error   := feedback.Error;
		stRtPartAllowEnable.ErrorID := feedback.ErrorId;
		stRtPartAllowEnable.stInfo  := stInfo;
		
		eState := E_MethodKeepAliveMotionSystem.eIdle;
		nState := 0;
		ccl_PartAllowEnable := TRUE;
		
	
	END_CASE

	feedback.Update();
END_METHOD

METHOD ccl_PartForceDisable : BOOL

VAR_INST
	
	nState			: INT;
	feedback		: MC_PlanarFeedback;
	stInfo			: ST_CommandReturnInfo;

END_VAR


	CASE nState OF
	
	0:
		part[PartToDisable].ForceDisable(feedback);
		
		stRtPartForceDisable.Active  := FALSE;
		stRtPartForceDisable.Busy    := FALSE;
		
		nState	:= 10;
		
		
	10:
		IF feedback.Done
		OR feedback.Error
		THEN
			nState := 100;
		END_IF
			
		
	100:  // Done or Error
		stInfo.nObjectID := feedback.objectInfo.Id;
		stInfo.nObjectType := feedback.objectInfo.ObjectType;
	
	
		stRtPartForceDisable.Aborted := FALSE;
		stRtPartForceDisable.Active  := FALSE;
		stRtPartForceDisable.Busy    := FALSE;
		stRtPartForceDisable.Done    := feedback.Done;
		stRtPartForceDisable.Error   := feedback.Error;
		stRtPartForceDisable.ErrorID := feedback.ErrorId;
		stRtPartForceDisable.stInfo  := stInfo;
		
		eState := E_MethodKeepAliveMotionSystem.eIdle;
		nState := 0;
		ccl_PartForceDisable := TRUE;
		
	
	END_CASE

	feedback.Update();
END_METHOD

METHOD ccl_PartForceEnable : BOOL

VAR_INST
	
	nState			: INT;
	feedback		: MC_PlanarFeedback;
	stInfo			: ST_CommandReturnInfo;

END_VAR


	CASE nState OF
	
	0:
		part[PartToEnableForce].ForceEnable(feedback);
		
		stRtPartForceEnable.Active  := FALSE;
		stRtPartForceEnable.Busy    := FALSE;
		
		nState	:= 10;
		
		
	10:
		IF feedback.Done
		OR feedback.Error
		THEN
			nState := 100;
		END_IF
			
		
	100:  // Done or Error
		stInfo.nObjectID   := feedback.objectInfo.Id;
		stInfo.nObjectType := feedback.objectInfo.ObjectType;
	
	
		stRtPartForceEnable.Aborted := FALSE;
		stRtPartForceEnable.Active  := FALSE;
		stRtPartForceEnable.Busy    := FALSE;
		stRtPartForceEnable.Done    := feedback.Done;
		stRtPartForceEnable.Error   := feedback.Error;
		stRtPartForceEnable.ErrorID := feedback.ErrorId;
		stRtPartForceEnable.stInfo  := stInfo;
		
		eState := E_MethodKeepAliveMotionSystem.eIdle;
		nState := 0;
		ccl_PartForceEnable := TRUE;
		
	END_CASE

	feedback.Update();
END_METHOD

METHOD ccl_PartInitialize : BOOL

VAR_INST
	

	nState			: INT;
	nPartIDint		: OTCID;
	feedback		: MC_PlanarFeedback;
	stInfo			: ST_CommandReturnInfo;

END_VAR


	CASE nState OF
		
	
	0:
		nPartIDint := PartToInitialze;
		part[1].Initialize(feedback, nPartIDint, environment);
		
		stRtPartInitialize.Active  := FALSE;
		stRtPartInitialize.Busy    := FALSE;
		
		nState	:= 10;
		
		
	10:
		IF feedback.Done
		OR feedback.Error
		THEN
			nState := 100;
		END_IF
			
		
	100:  // Done or Error
		stInfo.nObjectID := feedback.objectInfo.Id;
		stInfo.nObjectType := feedback.objectInfo.ObjectType;
	
	
		stRtPartInitialize.Aborted := FALSE;
		stRtPartInitialize.Active  := FALSE;
		stRtPartInitialize.Busy    := FALSE;
		stRtPartInitialize.Done    := feedback.Done;
		stRtPartInitialize.Error   := feedback.Error;
		stRtPartInitialize.ErrorID := feedback.ErrorId;
		stRtPartInitialize.stInfo  := stInfo;
		
		eState := E_MethodKeepAliveMotionSystem.eIdle;
		nState := 0;
		ccl_PartInitialize := TRUE;
		
	
	END_CASE

	feedback.Update();
END_METHOD

METHOD ccl_PartInitializeMulti : BOOL

VAR_INST
	

	nState			: INT;
	nPartIDint		: OTCID;
	feedback		: MC_PlanarFeedback;
	stInfo			: ST_CommandReturnInfo;
	nErrorSituation	: UDINT;
	
	nPartCounter	: PVOID;
	ptrPartID		: POINTER TO OTCID; 

END_VAR


	CASE nState OF
		
	
	0:	
		stRtPartInitializeMulti.Active  := TRUE;
		stRtPartInitializeMulti.Busy    := TRUE;		
		
		IF nPartCnt <= Params_XPlanar.maxNumberOfParts THEN
			nPartCounter := 0;
			      nState := 10;
		ELSE
			nErrorSituation := 1;
			nState := 110;
		END_IF

		
			
	10:
		nPartCounter := nPartCounter +1;
		IF nPartCounter <= nPartCnt THEN
			 ptrPartID := AddressArrayPartID + (nPartCounter -1)*4;
			nPartIDint := ptrPartID^;				
			nState := 20;
		ELSE
			nState := 100;
		END_IF
	

	20:
		part[nPartCounter].Initialize(feedback, nPartIDint, environment);
		nState	:= 30;
		
		
	30:
		IF feedback.Done THEN
			nState := 10;
		ELSIF feedback.Error THEN
			nErrorSituation := 2;
			nState := 110;
		END_IF
		
		
			
	100: // Done 
		stInfo.nObjectID := feedback.objectInfo.Id;
		stInfo.nObjectType := feedback.objectInfo.ObjectType;
	
	
		stRtPartInitializeMulti.Aborted := FALSE;
		stRtPartInitializeMulti.Active  := FALSE;
		stRtPartInitializeMulti.Busy    := FALSE;
		stRtPartInitializeMulti.Done    := feedback.Done;
		stRtPartInitializeMulti.Error   := feedback.Error;
		stRtPartInitializeMulti.ErrorID := feedback.ErrorId;
		stRtPartInitializeMulti.stInfo  := stInfo;
		
		nState := 200;
		

		
	110: // Error

		stRtPartInitializeMulti.Aborted := FALSE;
		stRtPartInitializeMulti.Active  := FALSE;
		stRtPartInitializeMulti.Busy    := FALSE;
		stRtPartInitializeMulti.Done    := FALSE;
		stRtPartInitializeMulti.Error   := TRUE;
		
		CASE nErrorSituation OF
			
		1:	// Parameter maxNumberOfParts is smaller then part count
			stRtPartInitializeMulti.ErrorID := nErrorSituation;
				
		2: // Error during initialization
			stRtPartInitializeMulti.ErrorID := feedback.ErrorId;
			stRtPartInitializeMulti.stInfo  := stInfo;	
		
		END_CASE
			
		nState := 200;
		
		
	200: // End
		eState := E_MethodKeepAliveMotionSystem.eIdle;
		nState := 0;
		ccl_PartInitializeMulti := TRUE;
			
	
	
	END_CASE

	feedback.Update();
END_METHOD

METHOD ccl_PartReset : BOOL

VAR_INST
	
	nState			: INT;
	nPartIDint		: UDINT;
	feedback		: MC_PlanarFeedback;
	stInfo			: ST_CommandReturnInfo;

END_VAR


	CASE nState OF
	
	0:
		part[PartToReset].Reset(feedback);
		
		stRtPartReset.Active  := FALSE;
		stRtPartReset.Busy    := FALSE;
		
		nState	:= 10;
		
		
	10:
		IF feedback.Done
		OR feedback.Error
		THEN
			nState := 100;
		END_IF
			
		
	100:  // Done or Error
		stInfo.nObjectID := feedback.objectInfo.Id;
		stInfo.nObjectType := feedback.objectInfo.ObjectType;
	
	
		stRtPartReset.Aborted := FALSE;
		stRtPartReset.Active  := FALSE;
		stRtPartReset.Busy    := FALSE;
		stRtPartReset.Done    := feedback.Done;
		stRtPartReset.Error   := feedback.Error;
		stRtPartReset.ErrorID := feedback.ErrorId;
		stRtPartReset.stInfo  := stInfo;
		
		eState := E_MethodKeepAliveMotionSystem.eIdle;
		nState := 0;
		ccl_PartReset := TRUE;
		
	
	END_CASE

	feedback.Update();
END_METHOD

METHOD PROTECTED ccl_RemoveEnvironmentFromGroup : BOOL


CASE nState OF

	0:  // Prepare
		stRtRemoveEnvironment.Aborted := FALSE;
		stRtRemoveEnvironment.Active  := TRUE;
		stRtRemoveEnvironment.Busy    := TRUE;
		stRtRemoveEnvironment.Done    := FALSE;
		stRtRemoveEnvironment.Error   := FALSE;
		stRtRemoveEnvironment.ErrorID := 0;
		stRtRemoveEnvironment.stInfo  := _stResultErrorInfoClear;

		nState := 10;
	
		
	10:  // Remove goup from environment	
		environment.RemoveFromGroup(cmdFeedback);		
		nState := 20;
		
		
	20:  // Checking feedback
				              _bResultDone := cmdFeedback.Done;
				             _bResultError := cmdFeedback.Error;
			               _nResultErrorID := cmdFeedback.ErrorId;
			  _stResultErrorInfo.nObjectID := cmdFeedback.objectInfo.Id;
			_stResultErrorInfo.nObjectType := cmdFeedback.objectInfo.ObjectType;

		IF _bResultDone OR _bResultError THEN
			nState := 100;	
		END_IF	
		
	
	100:  // Done
		stRtRemoveEnvironment.Aborted  := FALSE;
		stRtRemoveEnvironment.Active   := FALSE;
		stRtRemoveEnvironment.Busy     := FALSE;
		stRtRemoveEnvironment.Done     := _bResultDone;
		stRtRemoveEnvironment.Error	   := _bResultError;
		stRtRemoveEnvironment.ErrorID  := _nResultErrorID;
		stRtRemoveEnvironment.stInfo   := _stResultErrorInfo;
		
		eState := E_MethodKeepAliveMotionSystem.eIdle;
		nState := 0;	
		ccl_RemoveEnvironmentFromGroup := TRUE;
		
		
END_CASE
END_METHOD

METHOD PROTECTED ccl_RemoveMoverFromGroup : BOOL

VAR_INPUT
	ipMover		: I_XPlanarMoverStandard;
END_VAR

CASE nState OF
	

	0:  // Prepare 
		stRtRemoveMover.Aborted := FALSE;
		stRtRemoveMover.Active  := TRUE;
		stRtRemoveMover.Busy    := TRUE;
		stRtRemoveMover.Done    := FALSE;
		stRtRemoveMover.Error   := FALSE;
		stRtRemoveMover.ErrorID := 0;
		stRtRemoveMover.stInfo  := _stResultErrorInfoClear;

		nState := 10;
		
		
	10:  // Removing the mover from the group
		bError := FALSE;		
		 bDone := TRUE;
		IF ipMover <> 0 THEN
			IF ipMover.P_InGroup THEN		
				bDone := ipMover.RemoveFromGroup();
			END_IF
		ELSE
			 bDone := FALSE;
			bError := TRUE;
		END_IF

		IF bDone OR bError THEN
			nState := 20;
		END_IF
		
		
	20:  // Checking feedback
		IF bError THEN
				  _bResultDone := FALSE;
				 _bResultError := TRUE;
			   _nResultErrorID := 1;	// Empty input -> no mover to remove from group
			_stResultErrorInfo := _stResultErrorInfoClear;	
		ELSE
				  _bResultDone := ipMover.P_RemoveFromGroup.Done;
				 _bResultError := ipMover.P_RemoveFromGroup.Error;
			   _nResultErrorID := ipMover.P_RemoveFromGroup.ErrorID;
			_stResultErrorInfo := ipMover.P_RemoveFromGroup.stInfo;	
		END_IF		
		
		IF _bResultDone OR _bResultError THEN
			nState := 100;
		END_IF
		
	
	100:  // Done
		stRtRemoveMover.Aborted  := FALSE;
		stRtRemoveMover.Active   := FALSE;
		stRtRemoveMover.Busy     := FALSE;
		stRtRemoveMover.Done     := _bResultDone;
		stRtRemoveMover.Error    := _bResultError;
		stRtRemoveMover.ErrorID  := _nResultErrorID;
		stRtRemoveMover.stInfo   := _stResultErrorInfo;
		
		eState := E_MethodKeepAliveMotionSystem.eIdle;
		nState := 0;
		ccl_RemoveMoverFromGroup := TRUE;	


END_CASE
END_METHOD

METHOD PROTECTED ccl_RemoveMoversFromGroup : BOOL


CASE nState OF

	0:  // Prepare 
		stRtRemoveMovers.Aborted  := FALSE;
		stRtRemoveMovers.Active   := TRUE;
		stRtRemoveMovers.Busy     := TRUE;
		stRtRemoveMovers.Done     := FALSE;
		stRtRemoveMovers.Error    := FALSE;
		stRtRemoveMovers.ErrorID  := 0;
		stRtRemoveMovers.stInfo   := _stResultErrorInfoClear;

		nState := 10;
		
		
	10:  // Remove all movers from the group  
		bDone := TRUE;
		FOR nForCounter := 1 TO _nAxisCount DO
			IF ipMover[nForCounter] <> 0 THEN			
				IF ipMover[nForCounter].P_InGroup THEN		
					bDone := bDone AND ipMover[nForCounter].RemoveFromGroup();
				END_IF
			END_IF
		END_FOR
		
		IF bDone THEN
			nState := 20;
		END_IF
		
		
	20:  // Checking feedback	
		bError := FALSE;
		 bDone := TRUE;
		FOR nForCounter := 1 TO _nAxisCount DO
			IF NOT ipMover[nForCounter].P_InGroup THEN
				bDone := bDone AND TRUE;	
			ELSE
				bDone := FALSE;
				IF ipMover[nForCounter].P_RemoveFromGroup.Error THEN
					IF NOT bError THEN
						           bError := TRUE;
						         nErrorID := ipMover[nForCounter].P_RemoveFromGroup.ErrorID;
						stResultErrorInfo := ipMover[nForCounter].P_RemoveFromGroup.stInfo;
					END_IF
				END_IF
			END_IF
		END_FOR		
		
		IF bDone OR bError THEN
				  _bResultDone := bDone;
				 _bResultError := bError;
			   _nResultErrorID := nErrorID;
			_stResultErrorInfo := stResultErrorInfo;			
					
			nState := 100;	
		END_IF
		
		
	100:  // Done
		stRtRemoveMovers.Aborted  := FALSE;
		stRtRemoveMovers.Active   := FALSE;
		stRtRemoveMovers.Busy     := FALSE;
		stRtRemoveMovers.Done	  := _bResultDone;
		stRtRemoveMovers.Error    := _bResultError;
		stRtRemoveMovers.ErrorID  := _nResultErrorID;
		stRtRemoveMovers.stInfo   := _stResultErrorInfo;
	
		eState := E_MethodKeepAliveMotionSystem.eIdle;
		nState := 0;
		ccl_RemoveMoversFromGroup := TRUE;
			

END_CASE
END_METHOD

METHOD PROTECTED ccl_RemoveTracksFromGroup : BOOL



VAR_INST
	
	nTestCounter01	: UINT;
	
	nTrackToRemove	: INT;
	
END_VAR
CASE nState OF
	
	0:  // Prepare
		stRtRemoveTracks.Aborted  := FALSE;
		stRtRemoveTracks.Active   := TRUE;
		stRtRemoveTracks.Busy     := TRUE;
		stRtRemoveTracks.Done     := FALSE;
		stRtRemoveTracks.Error    := FALSE;
		stRtRemoveTracks.ErrorID  := 0;
		stRtRemoveTracks.stInfo   := _stResultErrorInfoClear;

		nState := 10;
		
		nTestCounter01 := nTestCounter01 +1;
	
		
		
		
	10: // Removing tracks from the group one-by-one
				    bDone := FALSE;
		           bError := FALSE;
		         nErrorID := 0;
		stResultErrorInfo := _stResultErrorInfoClear;
		   nTrackToRemove := 0;
		   
		nState := nState + 1;
	
	11: nTrackToRemove := nTrackToRemove +1;
		IF nTrackToRemove <= _nTrackCount THEN
			nState := nState + 1;
		ELSE
			 bDone := TRUE;
			nState := 20;
		END_IF
		
	12: IF ipTrack[nTrackToRemove].P_GroupOID <> 0 THEN
			nState := nState + 1;
		ELSE
			nState := nState - 1;
		END_IF 	
		
	13:	IF ipTrack[nTrackToRemove].RemoveFromGroup() THEN
			nState := nState + 1;
		END_IF
		
	14:	IF ipTrack[nTrackToRemove].P_RemoveFromGroup.Done THEN
			nState := nState - 3;
		ELSIF ipTrack[nTrackToRemove].P_RemoveFromGroup.Error THEN
				           bError := TRUE;
				         nErrorID := ipTrack[nForCounter].P_RemoveFromGroup.ErrorID;
				stResultErrorInfo := ipTrack[nForCounter].P_RemoveFromGroup.stInfo;			
				nState := 20;
		END_IF
		
		
	
	20: // Checking feedback 
		IF bDone OR bError THEN
			      _bResultDone := bDone;
			     _bResultError := bError;
			   _nResultErrorID := nErrorID;
			_stResultErrorInfo := stResultErrorInfo;
			            nState := 100;
		END_IF
		
	
	100:  // Done
		stRtRemoveTracks.Active  := FALSE;
		stRtRemoveTracks.Busy    := FALSE;
		stRtRemoveTracks.Done    := _bResultDone;
		stRtRemoveTracks.Error   := _bResultError;
		stRtRemoveTracks.ErrorID := _nResultErrorID;
		stRtRemoveTracks.stInfo  := _stResultErrorInfo;
		
		eState := E_MethodKeepAliveMotionSystem.eIdle;
		nState := 0;			   
		ccl_RemoveTracksFromGroup  := TRUE;

END_CASE
END_METHOD

METHOD PROTECTED ccl_ResetGroup : BOOL


CASE nState OF 

	0:  // Prepare 
		stRtResetGroup.Aborted  := FALSE;
		stRtResetGroup.Active   := TRUE;
		stRtResetGroup.Busy 	:= TRUE;
		stRtResetGroup.Done 	:= FALSE;
		stRtResetGroup.Error 	:= FALSE;
		stRtResetGroup.ErrorID 	:= 0; 
		stRtResetGroup.stInfo   := _stResultErrorInfoClear;
			
		nState := 10;
		
		
	10:  // Resetting the group
		Group.Reset(CmdFeedback);
		nState := 20;
		
		
	20:  // Checking feedback
			            _bResultDone := cmdFeedback.Done;
			           _bResultError := cmdFeedback.Error;
		             _nResultErrorID := cmdFeedback.ErrorId;
		_stResultErrorInfo.nObjectID := cmdFeedback.objectInfo.Id;			
		_stResultErrorInfo.nObjectID := cmdFeedback.objectInfo.ObjectType;	
			
		IF _bResultDone OR _bResultError THEN
			nState := 100;
		END_IF


	100:  // Done
		stRtResetGroup.Aborted  := FALSE;
		stRtResetGroup.Active   := FALSE;
		stRtResetGroup.Busy 	:= FALSE;
		stRtResetGroup.Done 	:= _bResultDone;
		stRtResetGroup.Error 	:= _bResultError;
		stRtResetGroup.ErrorID 	:= _nResultErrorID; 
		stRtResetGroup.stInfo   := _stResultErrorInfo;
	
		eState := E_MethodKeepAliveMotionSystem.eIdle;
		nState := 0; 
		ccl_ResetGroup := TRUE;
		
	
END_CASE
END_METHOD

METHOD PROTECTED ccl_ResetMovers : BOOL

VAR_INST
	CheckMoverState 	: MC_Planar_State;

	bResetCommandfeedback_Active  : BOOL;
	bResetCommandfeedback_Busy 	  : BOOL;
	bResetCommandfeedback_Done 	  : BOOL;
	bResetCommandfeedback_Error   : BOOL;
	nResetCommandfeedback_ErrorId : UDINT;
	stResetCommandfeedback_Info   : ST_CommandReturnInfo;
	
	sErrorLogMessage	: STRING;
END_VAR
CASE nState OF

	0:  // Prepare
		stRtResetMovers.Aborted  := FALSE;
		stRtResetMovers.Active   := TRUE;
		stRtResetMovers.Busy     := TRUE;
		stRtResetMovers.Done     := FALSE;
		stRtResetMovers.Error    := FALSE;
		stRtResetMovers.ErrorID	 := 0;
		stRtResetMovers.stInfo   := _stResultErrorInfoClear;
		
		nState := 10;
		
	
	10:  // Resetting all movers
		bDone := TRUE;
		FOR nForCounter := 1 TO _nAxisCount DO
			IF ipMover[nForCounter].P_State = MC_PLANAR_STATE.Error 
			OR ipMover[nForCounter].P_State = MC_PLANAR_STATE.ErrorPending
			OR ipMover[nForCounter].P_State = MC_PLANAR_STATE.Resetting
			THEN
				IF ipMover[nForCounter].P_State = MC_PLANAR_STATE.Error THEN
					sErrorLogMessage := 'Reset all movers - MoverState: Error';	
				ELSIF ipMover[nForCounter].P_State = MC_PLANAR_STATE.ErrorPending THEN
					sErrorLogMessage := 'Reset all movers - MoverState: ErrorPending';	
				
				ELSIF ipMover[nForCounter].P_State = MC_PLANAR_STATE.Resetting THEN
					sErrorLogMessage := 'Reset all movers - MoverState: Resetting';	
				END_IF
				bDone := bDone AND ipMover[nForCounter].Reset(sErrorLogMessage);
			END_IF			
		END_FOR
		IF bDone THEN
			nState := 20;
		END_IF
		
				
	20:  // Checking feedback
		bError := FALSE;
		 bDone := TRUE;
		FOR nForCounter := 1 TO _nAxisCount DO
			
			bResetCommandfeedback_Active  := ipMover[nForCounter].P_Reset.Active;
			bResetCommandfeedback_Busy 	  := ipMover[nForCounter].P_Reset.Busy;
			bResetCommandfeedback_Done 	  := ipMover[nForCounter].P_Reset.Done;
			bResetCommandfeedback_Error   := ipMover[nForCounter].P_Reset.Error;
			nResetCommandfeedback_ErrorId := ipMover[nForCounter].P_Reset.ErrorID;
			stResetCommandfeedback_Info   := ipMover[nForCounter].P_Reset.stInfo;
		
			IF ipMover[nForCounter].P_Reset.Done
			OR ipMover[nForCounter].P_Reset.Error
			THEN
				CheckMoverState := ipMover[nForCounter].P_State;
				IF CheckMoverState = MC_PLANAR_STATE.Error
				OR CheckMoverState = MC_PLANAR_STATE.ErrorPending
				OR CheckMoverState = MC_PLANAR_STATE.Resetting
				OR CheckMoverState = MC_PLANAR_STATE.Invalid
				THEN
					bDone := FALSE;
					IF ipMover[nForCounter].P_Reset.Error THEN
						IF NOT bError THEN
									   bError := TRUE;
									 nErrorID := nResetCommandfeedback_ErrorId;
							stResultErrorInfo := stResetCommandfeedback_Info;						
						END_IF
					ELSE
						(*
						// **** Repeat reset command
						IF ipMover[nForCounter].P_Reset.Done THEN
							nState := 10;
						END_IF
						*)
						EXIT;
					END_IF
				END_IF
			END_IF
		END_FOR
	
		IF bDone OR bError THEN
			      _bResultDone := bDone;
			     _bResultError := bError;
			   _nResultErrorID := nErrorID;			
			_stResultErrorInfo := stResultErrorInfo;		
	
			nState := 100;
		END_IF
	
		
	100:  // Done
		stRtResetMovers.Aborted  := FALSE;
		stRtResetMovers.Active   := FALSE;
		stRtResetMovers.Busy     := FALSE;
		stRtResetMovers.Done     := _bResultDone;
		stRtResetMovers.Error    := _bResultError;
		stRtResetMovers.ErrorID	 := _nResultErrorID;
		stRtResetMovers.stInfo   := _stResultErrorInfo;
	
		eState := E_MethodKeepAliveMotionSystem.eIdle;
		nState := 0;
		ccl_ResetMovers := TRUE;
		


END_CASE
END_METHOD

METHOD PROTECTED ccl_ResetParts : BOOL

VAR_INST
	CheckMoverState 	: MC_Planar_State;

	bResetCommandfeedback_Active  : BOOL;
	bResetCommandfeedback_Busy 	  : BOOL;
	bResetCommandfeedback_Done 	  : BOOL;
	bResetCommandfeedback_Error   : BOOL;
	nResetCommandfeedback_ErrorId : UDINT;
	stResetCommandfeedback_Info   : ST_CommandReturnInfo;
	
	sErrorLogMessage	: STRING;
	
	commandFB			: ARRAY [1..Params_XPlanar.maxNumberOfParts] OF MC_PlanarFeedback;
	

END_VAR
CASE nState OF

	0:  // Prepare
		stRtResetParts.Aborted  := FALSE;
		stRtResetParts.Active   := TRUE;
		stRtResetParts.Busy     := TRUE;
		stRtResetParts.Done     := FALSE;
		stRtResetParts.Error    := FALSE;
		stRtResetParts.ErrorID	:= 0;
		stRtResetParts.stInfo   := _stResultErrorInfoClear;
		
		nState := 10;
		
	
	10:  // Resetting all movers
		FOR idx := 1 TO Params_XPlanar.maxNumberOfParts DO
			IF part[idx].PartOID > 0 THEN
				part[idx].Reset(commandFB[idx]);
			END_IF
		END_FOR 
		nState := nState +10;
		
		
	20: // Checking the feedback
		nErrorID := 0;
		stResultErrorInfo := _stResultErrorInfoClear;
	
		 bDone := TRUE;
		bError := FALSE;
		FOR idx := 1 TO Params_XPlanar.maxNumberOfParts DO
			IF part[idx].PartOID > 0 THEN
				commandFB[idx].Update();	
			
			     bDone := bDone AND commandFB[idx].Done;
				bError := bError OR commandFB[idx].Error;
				
				IF bError THEN
					                     nErrorID := commandFB[idx].ErrorId;
					  stResultErrorInfo.nObjectID := commandFB[idx].objectInfo.Id;	
					stResultErrorInfo.nObjectType := commandFB[idx].objectInfo.ObjectType;
					EXIT;
				END_IF
			END_IF
		
		END_FOR 
		
		IF bDone OR bError THEN
			nState := 100;
		END_IF
		
				
	
	100:  // Done
		stRtResetParts.Aborted  := FALSE;
		stRtResetParts.Active   := FALSE;
		stRtResetParts.Busy     := FALSE;
		stRtResetParts.Done     := bDone;
		stRtResetParts.Error    := bError;
		stRtResetParts.ErrorID	:= nErrorID;
		stRtResetParts.stInfo   := stResultErrorInfo;
	
		eState := E_MethodKeepAliveMotionSystem.eIdle;
		nState := 0;
		ccl_ResetParts := TRUE;
		

END_CASE
END_METHOD

METHOD PROTECTED ccl_ResetTracks : BOOL

VAR_INST
	nTrackToReset	: DINT;
END_VAR

CASE nState OF 
	
	0:  // Prepare 
		stRtResetTracks.Aborted	:= FALSE;
		stRtResetTracks.Active  := TRUE;
		stRtResetTracks.Busy 	:= TRUE;
		stRtResetTracks.Done 	:= FALSE;;
		stRtResetTracks.Error 	:= FALSE;
		stRtResetTracks.ErrorID := 0; 
		stRtResetTracks.stInfo  := _stResultErrorInfoClear;
		
		nTrackToReset := 0;
		nState := 10;
		
		
	10:  // Reset all tracks one-by-one
		nTrackToReset := nTrackToReset +1;
		IF nTrackToReset <= _nTrackCount THEN
			IF ipTrack[nTrackToReset] <> 0 THEN
				nState := nState +1;
			END_IF
		ELSE
			// All tracks are resetted
						bDone := TRUE;		
					   bError := FALSE;				
					 nErrorID := 0;
			stResultErrorInfo := _stResultErrorInfoClear;
		
			nState := 100;
		END_IF
		
		
	11:	 // Check current track state, if necessary perform reset
		IF ipTrack[nTrackToReset].P_State = MC_Planar_State.Error
		OR ipTrack[nTrackToReset].P_State = MC_Planar_State.ErrorPending
		THEN
			IF ipTrack[nTrackToReset].Reset() THEN
				nState := nState +1;
			END_IF
		ELSE
			nState := nState -1;
		END_IF
		
		
	12:  // Check feedback
		            bDone := ipTrack[nTrackToReset].P_Reset.Done;				
		           bError := ipTrack[nTrackToReset].P_Reset.Error;				
		         nErrorID := ipTrack[nTrackToReset].P_Reset.ErrorID;
		stResultErrorInfo := ipTrack[nTrackToReset].P_Reset.stInfo;

		IF bDone THEN
			nState := 10;
		ELSIF bError THEN
			nState := 100;
		END_IF
		

		
	100:  //  Done
		stRtResetTracks.Aborted	:= FALSE;
		stRtResetTracks.Active  := FALSE;
		stRtResetTracks.Busy 	:= FALSE;
		stRtResetTracks.Done 	:= bDone;;
		stRtResetTracks.Error 	:= bError;
		stRtResetTracks.ErrorID := nErrorID; 
		stRtResetTracks.stInfo  := stResultErrorInfo;

		eState := E_MethodKeepAliveMotionSystem.eIdle;
		nState := 0;
		ccl_ResetTracks := TRUE;		
		
		

END_CASE
END_METHOD

METHOD PROTECTED ResetStateVariables : BOOL
VAR_INPUT
END_VAR
nState :=0;
END_METHOD

METHOD Cycle
VAR_INPUT
END_VAR
// Update of XPlanar logic



//IF bInit THEN
//    bInit := FALSE; 
//    fbMsg.CreateEx(TC_EVENTS.XPlanarStdLibEventClass.Check_01, 0); 
//END_IF

//IF bSend THEN 
//    bSend := FALSE; 
//    fbMsg.Send(0); 
//END_IF




ccl_MethodKeepAlive();
group.Update();
environment.Update();


CASE nStateInitXpu OF


0: 	nStateInitXpu := 1;
	

1: // init environment
	sInitInfo := 'Waiting for Environment initialization!';

	IF fbEnvironment.Init(TRUE) THEN
		fbEnvironment.Init(FALSE);
		sInitInfo := 'Environment initialized';
		nStateInitXpu := 10;
	END_IF

	
10: // init Visu
	fbVisuXPlanarDiag.Environment := fbEnvironment;
	nStateInitXpu := 20;
	
	
20: // init XPU
	IF nIndexXPU = 0 THEN
		nIndexXPU := 1;
	END_IF

	ipXpuInternal := fbEnvironment.XpuTcIo(nIndexXPU);
	
	IF ipXpuInternal <> 0 THEN
		nStateInitXpu := nStateInitXpu +1;
	ELSE
		sInitInfo := 'No XPU from Environment!';
	END_IF
	
21:
	sInitInfo := 'Initialization done.';
	bSystemInitialized := TRUE;
	nStateInitXpu := nStateInitXpu +1;
	
ELSE // call Visu
	fbVisuXPlanarDiag.Environment := fbEnvironment;
	fbVisuXPlanarDiag.Cycle();
END_CASE
END_METHOD

PROPERTY ipDriver : I_Environment
GET
ipDriver := fbEnvironment;
END_GET
END_PROPERTY

{attribute 'hide'}
PROPERTY ipTcIoMover : ARRAY [1..Params_XPlanar.maxNumMover] OF I_TcIoXPlanarMover;
GET
ipTcIoMover := ipTcIoXPlanarMover;
END_GET
END_PROPERTY

PROPERTY P_IndexXPU : UINT
GET
P_IndexXPU := nIndexXPU;
END_GET
SET
nIndexXPU := P_IndexXPU;
END_SET
END_PROPERTY

PROPERTY P_SystemInitialized : BOOL
GET
P_SystemInitialized := bSystemInitialized;
END_GET
END_PROPERTY

METHOD SetMoverStandard : I_XPlanarMoverStandard
VAR_INPUT
	nnum : UDINT;
	ipMoverStandard	: I_XPlanarMoverStandard;
END_VAR
VAR
	nCnt : UDINT;
END_VAR


IF nNum <= Params_XPlanar.maxNumMover THEN
	
	ipMover[nNum] := ipMoverStandard;
	
	_nAxisCount := 0;
	FOR nCnt := 1 TO Params_XPlanar.maxNumMover DO
		IF ipMover[nCnt] <> 0 THEN
			_nAxisCount := _nAxisCount +1;
		END_IF
	END_FOR

END_IF
END_METHOD

METHOD SetTrackStandard : Bool
VAR_INPUT
	nnum : UDINT;
	ipTrackStandard	: I_TrackStandard;
END_VAR
VAR
	nCnt : UDINT;
END_VAR


IF nNum <= Params_XPlanar.maxTrackCount THEN

	ipTrack[nNum] := ipTrackStandard;
	
	_nTrackCount := 0;
	FOR nCnt := 1 TO Params_XPlanar.maxTrackCount DO
		IF ipTrack[nCnt] <> 0 THEN
			_nTrackCount := _nTrackCount +1;
		END_IF
	END_FOR

END_IF
END_METHOD


{attribute 'hide'}
METHOD WriteParameter : DINT

VAR_INPUT
	oidObject  		: OTCID;
	pidParameter 	: PTCID;
	
	nDataSize		: UDINT;
	pData			: PVOID;
END_VAR

VAR_INST
	iTcComObj 					: ITComObject; 
	pOidExternalFeedback 		: POINTER TO OTCID; 
	hrResult					: HRESULT;
	
	nResult						: DINT;
END_VAR

			
	
	IF oidObject <> 0 THEN
		// This function returns an interface pointer to an object instance specified by means of object ID.
		hrResult := FW_ObjMgr_GetObjectInstance(	   oid := oidObject,
													   iid := TC_GLOBAL_IID_LIST.IID_ITComObject,
													pipUnk := ADR(iTcComObj)); 
													
		IF iTcComObj <> 0 THEN
			IF pidParameter <> 0 THEN
				
				hrResult := iTcComObj.TcSetObjPara(   pid := pidParameter, 
													nData := nDataSize, 
													pData := pData, 
													  pgp := 0); 
						  
				CASE hrResult OF
				s_OK: 					nResult := +1;
				s_FALSE:				nResult := -10;
				s_PENDING:				nResult := 0;
				S_WATCHDOG_TIMEOUT:		nResult := -11;
				E_FAIL:					nResult := -12;	
				ELSE	
					nResult := 0;
				END_CASE
				
			END_IF
		ELSE
			nResult := -2;
		END_IF
	ELSE
		nResult := -1;																														
	END_IF
								   
	WriteParameter := nResult;
END_METHOD

END_FUNCTION_BLOCK

// XPlanarStandardFunctions/MotionSystem/I_MotionSystem
INTERFACE I_MotionSystem EXTENDS __SYSTEM.IQueryInterface

PROPERTY P_AddEnviromentToGroup : REFERENCE TO ST_CommandReturn
GET
END_GET
END_PROPERTY

PROPERTY P_AddModuleToEnvironment : REFERENCE TO ST_CommandReturn
GET
END_GET
END_PROPERTY

PROPERTY P_AddMoversToGroup : REFERENCE TO ST_CommandReturn
GET
END_GET
END_PROPERTY

PROPERTY P_AddMoverToGroup : REFERENCE TO ST_CommandReturn
GET
END_GET
END_PROPERTY

PROPERTY P_AddTracksToGroup : REFERENCE TO ST_CommandReturn
GET
END_GET
END_PROPERTY

PROPERTY P_CheckValidMovers : REFERENCE TO ST_MoverCheckInfo
GET
END_GET
END_PROPERTY

PROPERTY P_DisableGroup : REFERENCE TO ST_CommandReturn
GET
END_GET
END_PROPERTY

PROPERTY P_DisableMovers : REFERENCE TO ST_CommandReturn
GET
END_GET
END_PROPERTY

PROPERTY P_DisableTracks : REFERENCE TO ST_CommandReturn
GET
END_GET
END_PROPERTY

PROPERTY P_EnableGroup : REFERENCE TO ST_CommandReturn
GET
END_GET
END_PROPERTY

PROPERTY P_EnableMovers : REFERENCE TO ST_CommandReturn
GET
END_GET
END_PROPERTY

PROPERTY P_EnableTrack : REFERENCE TO ST_CommandReturn
GET
END_GET
END_PROPERTY

PROPERTY P_EnableTracks : REFERENCE TO ST_CommandReturn
GET
END_GET
END_PROPERTY

PROPERTY P_HaltSystem : REFERENCE TO ST_CommandReturn
GET
END_GET
END_PROPERTY

PROPERTY P_LeaveTrack : REFERENCE TO ST_CommandReturn
GET
END_GET
END_PROPERTY

PROPERTY P_PartActivatePosition : REFERENCE TO ST_CommandReturn
GET
END_GET
END_PROPERTY

PROPERTY P_PartAllowEnable : REFERENCE TO ST_CommandReturn
GET
END_GET
END_PROPERTY

PROPERTY P_PartForceDisable : REFERENCE TO ST_CommandReturn
GET
END_GET
END_PROPERTY

PROPERTY P_PartInitialize : REFERENCE TO ST_CommandReturn
GET
END_GET
END_PROPERTY

PROPERTY P_PartInitializeMulti : REFERENCE TO ST_CommandReturn
GET
END_GET
END_PROPERTY

PROPERTY P_PartReset : REFERENCE TO ST_CommandReturn
GET
END_GET
END_PROPERTY

PROPERTY P_RemoveEnviromentFromGroup : REFERENCE TO ST_CommandReturn
GET
END_GET
END_PROPERTY

PROPERTY P_RemoveMoverFromGroup : REFERENCE TO ST_CommandReturn
GET
END_GET
END_PROPERTY

PROPERTY P_RemoveMoversFromGroup : REFERENCE TO ST_CommandReturn
GET
END_GET
END_PROPERTY

PROPERTY P_RemoveTracksFromGroup : REFERENCE TO ST_CommandReturn
GET
END_GET
END_PROPERTY

PROPERTY P_ResetGroup : REFERENCE TO ST_CommandReturn
GET
END_GET
END_PROPERTY

PROPERTY P_ResetMovers : REFERENCE TO ST_CommandReturn
GET
END_GET
END_PROPERTY

PROPERTY P_ResetParts : REFERENCE TO ST_CommandReturn
GET
END_GET
END_PROPERTY

PROPERTY P_ResetTracks : REFERENCE TO ST_CommandReturn
GET
END_GET
END_PROPERTY

METHOD AddEnvironmentToGroup : BOOL
END_METHOD

METHOD AddModuleToEnvironment : BOOL
VAR_INPUT
	xPos : LREAL;
	yPos : LREAL;
END_VAR
END_METHOD

METHOD AddMoversToGroup : BOOL
END_METHOD

METHOD AddMoverToGroup : BOOL
VAR_INPUT
	ipMover		: I_XPlanarMoverStandard;
END_VAR
END_METHOD

METHOD AddTracksToGroup : BOOL
END_METHOD

METHOD CheckValidMovers : BOOL
VAR_INPUT
END_VAR
END_METHOD

METHOD DisableGroup : BOOL
END_METHOD

METHOD DisableMovers : BOOL
END_METHOD

METHOD DisableTracks : BOOL
VAR_INPUT
END_VAR
END_METHOD

METHOD EnableGroup : BOOL
END_METHOD

METHOD EnableMovers : BOOL
END_METHOD

METHOD EnableTrack : BOOL
VAR_INPUT
	ipTrackToAdd	: I_TrackStandard;
END_VAR
END_METHOD

METHOD EnableTracks : BOOL
END_METHOD

METHOD HaltSystem : BOOL
END_METHOD

METHOD LeaveTrack : BOOL
END_METHOD

METHOD PartActivatePosition : BOOL
VAR_INPUT
	nPartIndex		: UINT;
	nPositionIndex	: UINT;
END_VAR
END_METHOD

METHOD PartAllowEnable : BOOL
VAR_INPUT
	nPartID		: UDINT;
END_VAR
END_METHOD

METHOD PartForceDisable : BOOL
VAR_INPUT
	nPartID		: UDINT;
END_VAR
END_METHOD

METHOD PartInitialize : BOOL
VAR_INPUT
	
	nPartID		: OTCID;


END_VAR
END_METHOD

METHOD PartInitializeMulti : BOOL
VAR_INPUT
	
	AdrPartID		: PVOID;
	nPartCount		: UINT;
	
END_VAR
END_METHOD

METHOD PartReset : BOOL
VAR_INPUT
	nPartID		: UDINT;
END_VAR
END_METHOD

METHOD RemoveEnvironmentFromGroup : BOOL
END_METHOD

METHOD RemoveMoverFromGroup : BOOL
VAR_INPUT
	ipMover		: I_XPlanarMoverStandard;
END_VAR
END_METHOD

METHOD RemoveMoversFromGroup : BOOL
END_METHOD

METHOD RemoveTracksFromGroup : BOOL
END_METHOD

METHOD ResetGroup : BOOL
END_METHOD

METHOD ResetMovers : BOOL
END_METHOD

METHOD ResetParts : BOOL
END_METHOD

METHOD ResetTracks : BOOL
END_METHOD

METHOD UtilityCheckForError : DINT
VAR_INPUT
	bAutoReset : BOOL;
END_VAR
END_METHOD

METHOD UtilityErrorReset : BOOL
VAR_INPUT
END_VAR
END_METHOD

METHOD Cycle
END_METHOD


PROPERTY ipDriver : I_Environment
GET
END_GET
END_PROPERTY

PROPERTY P_IndexXPU : UINT
GET
END_GET
SET
END_SET
END_PROPERTY

PROPERTY P_SystemInitialized : BOOL
GET
END_GET
END_PROPERTY

METHOD SetMoverStandard : I_XPlanarMoverStandard
VAR_INPUT
	nnum : UDINT;
	ipMoverStandard	: I_XPlanarMoverStandard;
END_VAR
END_METHOD

METHOD SetTrackStandard : Bool
VAR_INPUT
	nnum : UDINT;
	ipTrackStandard	: I_TrackStandard;
END_VAR
END_METHOD


{attribute 'hide'}
METHOD WriteParameter : DINT

VAR_INPUT
	oidObject  		: OTCID;
	pidParameter 	: PTCID;
	
	nDataSize		: UDINT;
	pData			: PVOID;
END_VAR
END_METHOD

END_INTERFACE

// XPlanarStandardFunctions/Mover/BaseFunctions/MoverVectorToPostionXYC
FUNCTION MoverVectorToPostionXYC : REFERENCE TO PositionXYC
VAR_INPUT
	stPosMoverVector	: MOverVector;
END_VAR
VAR
	postion 		: PositionXYC;
END_VAR

	postion.SetValuesXYC(stPosMoverVector.x,stPosMoverVector.y,stPosMoverVector.c);
	
	MoverVectorToPostionXYC REF= postion;

END_FUNCTION

// XPlanarStandardFunctions/Mover/Experimental/FB_MoverTarget
{attribute 'hide'}
FUNCTION_BLOCK FB_MoverTarget
VAR_INPUT
END_VAR
VAR_OUTPUT
END_VAR
VAR
	
	positionList		: ARRAY[1..MaxMovers] OF ST_PositionXY;
	nPositionCount		: UDINT;
	moverList			: ARRAY[1..MaxMovers] OF I_MoverApplication;	
	nMoversInList		: UDINT;
	
	nErrorWarningCode 	: DINT;
	sMessage 			: STRING;
	
	idx					: UDINT;
	
	recoverVelocity					: LREAL :=   250.0;
	recoveryAcceleration			: LREAL :=  1000.0;
	recoveryJerk					: LREAL := 10000.0;
	
	nStateMove						: DINT;
END_VAR




// This function block can be used to move movers to pre-defined positions.
// The function block is experimental and worked well for tested scenarios on the starterkit application.
// It might work on other applications as well. If not it can be easily adapted since the code is open to edit.
// If you adapt this code to your machine's needs we're happy to hear from you to improve this function block for the XPlanar-Community.

METHOD AddMover : BOOL
VAR_INPUT
	ipMover		: I_MoverApplication;
END_VAR



VAR
	bMoverInList	: BOOL;
END_VAR


	IF ipMover <> 0 THEN
	
		nMoversInList := 0;
		bMoverInList  := FALSE;
		FOR idx:=1 TO nMoverCount DO
			IF moverList[idx] <> 0 THEN
				nMoversInList := nMoversInList +1;
				IF moverList[idx].std.P_Id = ipMover.std.P_Id THEN
					bMoverInList := TRUE;
				END_IF				
			END_IF
		END_FOR
		
		IF NOT bMoverInList THEN
			nMoversInList := nMoversInList +1;
			moverList[nMoversInList] := ipMover;
			
			nErrorWarningCode := 0;
		            sMessage := 'Success: Mover added.';				
		ELSE
			nErrorWarningCode := +11;
		            sMessage := 'Warning: Mover already exists.';				
		END_IF

	ELSE
		nErrorWarningCode := -11;
		        sMessage := 'Error: Mover invalid';	
	END_IF
	
	IF nErrorWarningCode < 0 THEN
		AddMover := FALSE;
	ELSE
		AddMover := TRUE;
	END_IF
END_METHOD

METHOD AddPosition : BOOL
VAR_INPUT
	x 	: LREAL;
	y	: LREAL;	
END_VAR



	nPositionCount := nPositionCount +1;
	
	IF nPositionCount <= nMoverCount THEN
	
		positionList[nPositionCount].x     := x;
		positionList[nPositionCount].y     := y;
		positionList[nPositionCount].valid := TRUE;

		nErrorWarningCode := 0;
		        sMessage := 'Success: Position added.';				
	ELSE
		nPositionCount := nMoverCount;	
	
		nErrorWarningCode := -21;
		        sMessage := 'Error: Position count higher than mover count!';				
	END_IF

	IF nErrorWarningCode < 0 THEN
		AddPosition := FALSE;
	ELSE
		AddPosition := TRUE;
	END_IF
END_METHOD

METHOD Clear : BOOL
VAR_INPUT
END_VAR




	FOR idx:=1 TO nMoverCount DO
		MoverList[idx] := 0;
		
		positionList[idx].x     := 0;
		positionList[idx].y     := 0;
		positionList[idx].valid := FALSE;
		
	END_FOR	
	
	    nMoversInList := 0;
	   nPositionCount := 0;	
	       nStateMove := 0;
	nErrorWarningCode := 0;
			sMessage := 'Cleared';				

	Clear := TRUE;
END_METHOD

METHOD MoversToTarget : BOOL
VAR_INPUT
END_VAR



VAR_INST
	
	idx1, idx2						: UDINT;
	idxMover, idxPosition			: UDINT;
	fShortestDistance				: LREAL;
	targetPosition					: PositionXYC;
	currentPos						: PositionXYC;
	bDone							: BOOL;	
	
	fMoverDistanceToInitialPosition	: ARRAY [1..MaxMovers, 1..MaxMovers] OF ST_MoverDistance;   // Mover;Position
	nMoverToInitialPosition			: ARRAY [1..MaxMovers] OF UDINT;
	nInitialPositionTakesMover		: ARRAY [1..MaxMovers] OF UDINT;
	nMoveStatus						: ARRAY [1..MaxMovers] OF DINT;
	nInitialPositionTaken			: ARRAY [1..MaxMovers] OF BOOL;	
	nInitialMoverTaken				: ARRAY [1..MaxMovers] OF BOOL;	
	nMoverTaken						: UDINT;
	bMovetToPositionXYC				: BOOL;
	
	fShiftDistanceY			: LREAL := 113.0;
	fShiftDistanceX			: LREAL := 113.0;
	
	
END_VAR


VAR_INST
	bMover01_Error 		: BOOL;
	bMover02_Error 		: BOOL;
	
	stInfoMover01		: ST_CommandReturnInfo;
	stInfoMover02		: ST_CommandReturnInfo;
	

	

END_VAR
	
	CASE nStateMove OF 
		
	
	0:	// Check mover and position count
		IF nMoversInList <= nPositionCount THEN
			nErrorWarningCode := 0;
			        sMessage := 'Mover and position count OK.';	
			      nStateMove := nStateMove + 10;
		ELSE
			nErrorWarningCode := -31;
					sMessage := 'Error: Mover count higher than position count!';				
		END_IF
	
		
	10:	// Clear 
		FOR idx:=1 TO nMoverCount DO
			        nMoveStatus[idx] := 0;
			 nInitialMoverTaken[idx] := 0;
		END_FOR	
		nStateMove := nStateMove + 10;
		
	
	20: // Calculate all distances
		FOR idx1:=1 TO nMoverCount DO
			FOR idx2:=1 TO nMoverCount DO
				fMoverDistanceToInitialPosition[idx1, idx2].fDistance      := 0.0;
				fMoverDistanceToInitialPosition[idx1, idx2].nPositionIndex := 0;
			END_FOR
		END_FOR
	
	
		FOR idx1:=1 TO nMoversInList DO
			currentPos.SetValuesXYC(moverList[idx1].std.P_SetPosition.x, moverList[idx1].std.P_SetPosition.y, moverList[idx1].std.P_SetPosition.c);
			FOR idx2:=1 TO nPositionCount DO
				fMoverDistanceToInitialPosition[idx1, idx2].nPositionIndex := idx2;		
				fMoverDistanceToInitialPosition[idx1, idx2].fDistance := SQRT((currentPos.x - positionList[idx2].x) * (currentPos.x - positionList[idx2].x) + (currentPos.y - positionList[idx2].y) * (currentPos.y - positionList[idx2].y)); 
			END_FOR	
			
			nInitialPositionTaken[idx1] := FALSE;
		END_FOR			

		nErrorWarningCode := 0;
				sMessage := 'Calculated all distances.';			
		      nStateMove := nStateMove + 10;
	
		
	30: // Find the closest initial position for each mover	
		FOR idxPosition:=1 TO nPositionCount DO
			fShortestDistance := 1.7976931348623158E+308;
			FOR idxMover:=1 TO nMoversInList DO			
				IF NOT nInitialMoverTaken[idxMover] THEN
					IF fMoverDistanceToInitialPosition[idxMover, idxPosition].fDistance < fShortestDistance THEN
						fShortestDistance := fMoverDistanceToInitialPosition[idxMover, idxPosition].fDistance;
						nInitialPositionTakesMover[idxPosition] := idxMover;
						nMoverTaken := idxMover;
					END_IF
				END_IF
			END_FOR
			IF nMoverTaken > 0 THEN
				nInitialMoverTaken[nMoverTaken] := TRUE;
			END_IF
		END_FOR
		
		
		FOR idx:=1 TO nMoverCount DO
			nMoverToInitialPosition[nInitialPositionTakesMover[idx]] := idx;	
		END_FOR

		nErrorWarningCode := 0;
				sMessage := 'Calculated closest initial position for each mover.';			
		nStateMove := nStateMove + 10;
		
		
		
	40: // Turn all movers back to 0° 
		
		// -> warten auf Set-C rotation Feature aus der NC
			
		nStateMove := nStateMove + 10;
		
		
		
	50: // Moving all movers to their initial position

		nErrorWarningCode := 0;
				sMessage := 'Moving.';		
	
		FOR idx1:=1 TO nMoversInList DO
		
			// 1st: try direct move
			IF nMoveStatus[idx1] = 0 THEN
				currentPos.SetValuesXYC(moverList[idx1].std.P_SetPosition.x, moverList[idx1].std.P_SetPosition.y, moverList[idx1].std.P_SetPosition.c);
				targetPosition.SetValuesXYC(positionList[nMoverToInitialPosition[idx1]].x, positionList[nMoverToInitialPosition[idx1]].y, currentPos.c);
				moverList[idx1].std.MoveToPosition('ToTarget move direct', targetPosition, recoverVelocity, recoveryAcceleration, recoveryAcceleration, recoveryJerk);
				bMovetToPositionXYC := FALSE;
				nMoveStatus[idx1] := 1;
			END_IF
			
			
//			bMover01_Error := moverList[1].std.P_MoveToPositionXYC.Error; 
//			 stInfoMover01 := moverList[1].std.P_MoveToPosition.stInfo;
			
//			bMover02_Error := moverList[2].std.P_MoveToPosition.Error; 
//			 stInfoMover02 := moverList[2].std.P_MoveToPosition.stInfo;
			
			
			// 2nd: try direct move XYC
			IF nMoveStatus[idx1] = 1 THEN
				IF moverList[idx1].std.P_MoveToPosition.Error THEN
					currentPos.SetValuesXYC(moverList[idx1].std.P_SetPosition.x, moverList[idx1].std.P_SetPosition.y, moverList[idx1].std.P_SetPosition.c);
					targetPosition.SetValuesXYC(positionList[nMoverToInitialPosition[idx1]].x, positionList[nMoverToInitialPosition[idx1]].y, currentPos.c);
					moverList[idx1].std.MoveToPositionXYC('ToTarget move direct', targetPosition, recoverVelocity, recoveryAcceleration, recoveryAcceleration, recoveryJerk);
					bMovetToPositionXYC := TRUE;
					nMoveStatus[idx1] := 2;
				END_IF
			END_IF			
			
			// 3rd: try move in x-direction
			IF nMoveStatus[idx1] = 2 THEN
				IF moverList[idx1].std.P_MoveToPositionXYC.Error THEN
					IF moverList[idx1].std.P_SetPosition.x <> positionList[nMoverToInitialPosition[idx1]].x THEN
						currentPos.SetValuesXYC(moverList[idx1].std.P_SetPosition.x, moverList[idx1].std.P_SetPosition.y, moverList[idx1].std.P_SetPosition.c);
						targetPosition.SetValuesXYC(positionList[nMoverToInitialPosition[idx1]].x, currentPos.y, currentPos.c);
						moverList[idx1].std.MoveToPosition('ToTarget move in x', targetPosition, recoverVelocity, recoveryAcceleration, recoveryAcceleration, recoveryJerk);
						bMovetToPositionXYC := FALSE;
					END_IF
					nMoveStatus[idx1] := 3;
				END_IF
			END_IF
						
			// 4th: try move XYC in x-direction
			IF nMoveStatus[idx1] = 3 THEN
				IF moverList[idx1].std.P_MoveToPosition.Error THEN
					IF moverList[idx1].std.P_SetPosition.x <> positionList[nMoverToInitialPosition[idx1]].x THEN
						currentPos.SetValuesXYC(moverList[idx1].std.P_SetPosition.x, moverList[idx1].std.P_SetPosition.y, moverList[idx1].std.P_SetPosition.c);
						targetPosition.SetValuesXYC(positionList[nMoverToInitialPosition[idx1]].x, currentPos.y, currentPos.c);
						moverList[idx1].std.MoveToPositionXYC('ToTarget move in x', targetPosition, recoverVelocity, recoveryAcceleration, recoveryAcceleration, recoveryJerk);
						bMovetToPositionXYC := TRUE;
					END_IF
					nMoveStatus[idx1] := 4;
				END_IF
			END_IF			
			
			// 5th: try move in y-direction
			IF nMoveStatus[idx1] = 4 THEN
				IF moverList[idx1].std.P_MoveToPositionXYC.Error THEN
					IF moverList[idx1].std.P_SetPosition.y <> positionList[nMoverToInitialPosition[idx1]].y THEN
						currentPos.SetValuesXYC(moverList[idx1].std.P_SetPosition.x, moverList[idx1].std.P_SetPosition.y, moverList[idx1].std.P_SetPosition.c);
						targetPosition.SetValuesXYC(currentPos.x, positionList[nMoverToInitialPosition[idx1]].y, currentPos.c);
						moverList[idx1].std.MoveToPosition('ToTarget move in y', targetPosition, recoverVelocity, recoveryAcceleration, recoveryAcceleration, recoveryJerk);
						bMovetToPositionXYC := FALSE;
					END_IF
					nMoveStatus[idx1] := 5; 
				END_IF		
			END_IF			
			
			// 6th: try move XYC in y-direction
			IF nMoveStatus[idx1] = 5 THEN
				IF moverList[idx1].std.P_MoveToPosition.Error THEN
					IF moverList[idx1].std.P_SetPosition.y <> positionList[nMoverToInitialPosition[idx1]].y THEN
						currentPos.SetValuesXYC(moverList[idx1].std.P_SetPosition.x, moverList[idx1].std.P_SetPosition.y, moverList[idx1].std.P_SetPosition.c);
						targetPosition.SetValuesXYC(currentPos.x, positionList[nMoverToInitialPosition[idx1]].y, currentPos.c);
						moverList[idx1].std.MoveToPositionXYC('ToTarget move in y', targetPosition, recoverVelocity, recoveryAcceleration, recoveryAcceleration, recoveryJerk);
						bMovetToPositionXYC := TRUE;
					END_IF
					nMoveStatus[idx1] := 6; 
				END_IF		
			END_IF				
			
			// 7th: try positive step-move in y-direction
			IF nMoveStatus[idx1] = 6 THEN
				IF moverList[idx1].std.P_MoveToPositionXYC.Error THEN
					currentPos.SetValuesXYC(moverList[idx1].std.P_SetPosition.x, moverList[idx1].std.P_SetPosition.y, moverList[idx1].std.P_SetPosition.c);
					targetPosition.SetValuesXYC(currentPos.x, currentPos.y + fShiftDistanceY, currentPos.c);
					moverList[idx1].std.MoveToPosition('ToTarget step-move in +y', targetPosition, recoverVelocity, recoveryAcceleration, recoveryAcceleration, recoveryJerk);
					bMovetToPositionXYC := FALSE;
					nMoveStatus[idx1] := 7; 
				END_IF		
			END_IF					
			
			// 8th: try positive step-move XYC in y-direction
			IF nMoveStatus[idx1] = 7 THEN
				IF moverList[idx1].std.P_MoveToPosition.Error THEN
					currentPos.SetValuesXYC(moverList[idx1].std.P_SetPosition.x, moverList[idx1].std.P_SetPosition.y, moverList[idx1].std.P_SetPosition.c);
					targetPosition.SetValuesXYC(currentPos.x, currentPos.y + fShiftDistanceY, currentPos.c);
					moverList[idx1].std.MoveToPositionXYC('ToTarget step-move in +y', targetPosition, recoverVelocity, recoveryAcceleration, recoveryAcceleration, recoveryJerk);
					bMovetToPositionXYC := TRUE;
					nMoveStatus[idx1] := 8; 
				END_IF		
			END_IF			
			
			// 9th: try negative step-move in y-direction
			IF nMoveStatus[idx1] = 8 THEN
				IF moverList[idx1].std.P_MoveToPositionXYC.Error THEN
					currentPos.SetValuesXYC(moverList[idx1].std.P_SetPosition.x, moverList[idx1].std.P_SetPosition.y, moverList[idx1].std.P_SetPosition.c);
					targetPosition.SetValuesXYC(currentPos.x, currentPos.y - fShiftDistanceX, currentPos.c);
					moverList[idx1].std.MoveToPosition('ToTarget step-move in -y', targetPosition, recoverVelocity, recoveryAcceleration, recoveryAcceleration, recoveryJerk);
					bMovetToPositionXYC := FALSE;
					nMoveStatus[idx1] := 9; 
				END_IF		
			END_IF	

			// 10th: try negative step-move XYC in y-direction
			IF nMoveStatus[idx1] = 9 THEN
				IF moverList[idx1].std.P_MoveToPosition.Error THEN
					currentPos.SetValuesXYC(moverList[idx1].std.P_SetPosition.x, moverList[idx1].std.P_SetPosition.y, moverList[idx1].std.P_SetPosition.c);
					targetPosition.SetValuesXYC(currentPos.x, currentPos.y - fShiftDistanceX, currentPos.c);
					moverList[idx1].std.MoveToPositionXYC('ToTarget step-move in -y', targetPosition, recoverVelocity, recoveryAcceleration, recoveryAcceleration, recoveryJerk);
					bMovetToPositionXYC := TRUE;
					nMoveStatus[idx1] := 10; 
				END_IF		
			END_IF		

			// 11th: try positive step-move in x-direction
			IF nMoveStatus[idx1] = 10 THEN
				IF moverList[idx1].std.P_MoveToPositionXYC.Error THEN
					currentPos.SetValuesXYC(moverList[idx1].std.P_SetPosition.x, moverList[idx1].std.P_SetPosition.y, moverList[idx1].std.P_SetPosition.c);
					targetPosition.SetValuesXYC(currentPos.x  + fShiftDistanceY, currentPos.y, currentPos.c);
					moverList[idx1].std.MoveToPosition('ToTarget step-move in +x', targetPosition, recoverVelocity, recoveryAcceleration, recoveryAcceleration, recoveryJerk);
					bMovetToPositionXYC := FALSE;
					nMoveStatus[idx1] := 11; 
				END_IF		
			END_IF	
			
			// 12th: try positive step-move XYC in x-direction
			IF nMoveStatus[idx1] = 11 THEN
				IF moverList[idx1].std.P_MoveToPosition.Error THEN
					currentPos.SetValuesXYC(moverList[idx1].std.P_SetPosition.x, moverList[idx1].std.P_SetPosition.y, moverList[idx1].std.P_SetPosition.c);
					targetPosition.SetValuesXYC(currentPos.x  + fShiftDistanceY, currentPos.y, currentPos.c);
					moverList[idx1].std.MoveToPositionXYC('ToTarget step-move in +x', targetPosition, recoverVelocity, recoveryAcceleration, recoveryAcceleration, recoveryJerk);
					bMovetToPositionXYC := TRUE;
					nMoveStatus[idx1] := 12; 
				END_IF		
			END_IF					
			
			// 13th: try negative step-move in x-direction
			IF nMoveStatus[idx1] = 12 THEN
				IF moverList[idx1].std.P_MoveToPositionXYC.Error THEN
					currentPos.SetValuesXYC(moverList[idx1].std.P_SetPosition.x, moverList[idx1].std.P_SetPosition.y, moverList[idx1].std.P_SetPosition.c);
					targetPosition.SetValuesXYC(currentPos.x - fShiftDistanceY, currentPos.y, currentPos.c);
					moverList[idx1].std.MoveToPosition('ToTarget step-move in -x', targetPosition, recoverVelocity, recoveryAcceleration, recoveryAcceleration, recoveryJerk);
					bMovetToPositionXYC := FALSE;
					nMoveStatus[idx1] := 13; 
				END_IF		
			END_IF				
			
			// 13th: try negative step-move XYC in x-direction
			IF nMoveStatus[idx1] = 13 THEN
				IF moverList[idx1].std.P_MoveToPosition.Error THEN
					currentPos.SetValuesXYC(moverList[idx1].std.P_SetPosition.x, moverList[idx1].std.P_SetPosition.y, moverList[idx1].std.P_SetPosition.c);
					targetPosition.SetValuesXYC(currentPos.x - fShiftDistanceY, currentPos.y, currentPos.c);
					moverList[idx1].std.MoveToPositionXYC('ToTarget step-move in -x', targetPosition, recoverVelocity, recoveryAcceleration, recoveryAcceleration, recoveryJerk);
										bMovetToPositionXYC := TRUE;
					nMoveStatus[idx1] := 14; 
				END_IF		
			END_IF				
			
			
			
			// Check feedback
			IF nMoveStatus[idx1] = 1 THEN
				IF moverList[idx1].std.P_MoveToPosition.Done THEN
					nMoveStatus[idx1] := 100;
				END_IF
			ELSIF nMoveStatus[idx1] = 2 THEN
				IF moverList[idx1].std.P_MoveToPositionXYC.Done THEN
					nMoveStatus[idx1] := 100;
				END_IF
			ELSE
				IF nMoveStatus[idx1] <> 100 THEN
					// If y-move is finished or no move was possible
					IF bMovetToPositionXYC THEN
						IF moverList[idx1].std.P_MoveToPositionXYC.Done
						OR moverList[idx1].std.P_MoveToPositionXYC.Error
						THEN
							nMoveStatus[idx1] := 0; 
						END_IF								
					ELSE
						IF moverList[idx1].std.P_MoveToPosition.Done
						OR moverList[idx1].std.P_MoveToPosition.Error
						THEN
							nMoveStatus[idx1] := 0; 
						END_IF						
					END_IF
				END_IF
			END_IF
			
			
		END_FOR
		
	
		// Check if all movers have reached their position
		bDone := TRUE;
		FOR idx1:=1 TO nMoversInList DO
			IF nMoveStatus[idx1] <> 100 THEN
				bDone := FALSE;
			END_IF
		END_FOR
			
		IF bDone THEN
			nStateMove := nStateMove + 10;
		END_IF
		

	60: // Done
		nErrorWarningCode := 0;
				sMessage := 'Done';			
	
		   nStateMove := 0;
		MoversToTarget := TRUE;
			
	END_CASE
END_METHOD

PROPERTY P_ErrorWarningCode : DINT
GET
P_ErrorWarningCode := nErrorWarningCode;
END_GET
END_PROPERTY

PROPERTY P_Info : STRING
GET
P_Info := sMessage;
END_GET
END_PROPERTY

METHOD SetDynamics : BOOL
VAR_INPUT
	vel	: LREAL;
	acc : LREAL;
	jerk :LREAL;
END_VAR

	recoverVelocity := vel;
	recoveryAcceleration := acc;
	recoveryJerk := jerk;
	
	SetDynamics := TRUE;
END_METHOD

END_FUNCTION_BLOCK

// XPlanarStandardFunctions/Mover/FB_XPlanarMoverStandard
FUNCTION_BLOCK FB_XPlanarMoverStandard IMPLEMENTS I_XPlanarMoverStandard
VAR_INPUT
END_VAR
VAR_OUTPUT
END_VAR
VAR
	stMoverRef 				: MC_PlanarMover;
	nId						: UINT;
	bInitHaltDynamicsDone	: BOOL;
	stHaltDynamics			: ST_HaltDynamics;
	
	ActPos 					: MoverVector;
	ActVelo					: MoverVector;
	SetPos 					: MoverVector;
	SetVelo 				: MoverVector;
	SetAcc 					: MoverVector;	
	SetOnTrack 				: CDT_MCTOPLC_PLANAR_MOVER_TRACK;
	nTrackId				: UDINT;	

	CurrentPosition			: MoverVector;	
	CurrentVelocity 		: MoverVector;	
	fCurrentAngleC			: LREAL;
 	fCurrentAngleC_Modulo	: LREAL;
	fClosestQuaterAngle		: LREAL;
	
	bIsSetpointGeneratorActive	: BOOL;
	bAtRotationPoint			: BOOL;
	bCRotationRestrictions		: BOOL;		
	bInGroup					: BOOL;
	bIsQueuing					: BOOL;
	bIsMovingXY					: BOOL;
	fZeroVelocityThreshold		: LREAL := 0.1;
	
	
	// store last MoveOnTrack Command
	stMoveOnTrackParameter		:  ST_MoveOnTrackParameters;
	
	CustomTrackIdTable			: ARRAY [1..Params_XPlanar.maxTrackCount] OF ST_CutomTrackID;


	
	// Command feedback	
	enableCmdFB 						: MC_PlanarFeedback;
	{attribute 'hide'}
	stRtEnable							: ST_CommandReturn;
	disableCmdFB 						: MC_PlanarFeedback;
	{attribute 'hide'}
	stRtDisable							: ST_CommandReturn;
	joinTrackCmdFB 						: MC_PlanarFeedback;
	{attribute 'hide'}
	stRtJoinTrack						: ST_CommandReturn;
	leaveTrackCmdFB 					: MC_PlanarFeedback;
	leaveTrackInPositionCmdFB 			: MC_PlanarFeedback;
	{attribute 'hide'}
	stRtLeaveTrack						: ST_CommandReturn;
	{attribute 'hide'}
	stRtLeaveTrackInPosition			: ST_CommandReturn;	
	moveOnTrackCmdFB 					: MC_PlanarFeedback;
	{attribute 'hide'}
	stRtMoveOnTrack						: ST_CommandReturn;
	{attribute 'hide'}
	stRtMoveOnTrackExt					: ST_CommandReturn;	
	moveOnTrackExtCmdFB 				: MC_PlanarFeedback;
		
	moveToPosCmdFB 						: MC_PlanarFeedback;
	{attribute 'hide'}
	stRtMoveToPos						: ST_CommandReturn;
	moveToPosXYCCmdFB 					: MC_PlanarFeedback;
	{attribute 'hide'}
	stRtMoveToPosXYC					: ST_CommandReturn;	
	moveToPosExtCmdFB 					: MC_PlanarFeedback;
	{attribute 'hide'}
	stRtMoveToPosExt					: ST_CommandReturn;		
	haltCmdFB 							: MC_PlanarFeedback;
	{attribute 'hide'}
	stRtHalt							: ST_CommandReturn;
	addMoverCmdFB						: MC_PlanarFeedback;
	{attribute 'hide'}
	stRtAddMover						: ST_CommandReturn;
	removeMoverCmdFB					: MC_PlanarFeedback;
	{attribute 'hide'}
	stRtRemoveMover						: ST_CommandReturn;
	resetCmdFB							: MC_PlanarFeedback;
	{attribute 'hide'}
	stRtReset							: ST_CommandReturn;
	moveZCmdFB							: MC_PlanarFeedback;
	{attribute 'hide'}
	stRtMoveZ							: ST_CommandReturn;
	moveACmdFB							: MC_PlanarFeedback;
	{attribute 'hide'}
	stRtMoveA							: ST_CommandReturn;
	moveBCmdFB							: MC_PlanarFeedback;
	{attribute 'hide'}
	stRtMoveB							: ST_CommandReturn;
	enableExtSetPosCmdFB				: MC_PlanarFeedback;
	{attribute 'hide'}
	stRtEnableSetPos					: ST_CommandReturn;
	disableExtSetPosCmdFB				: MC_PlanarFeedback;
	{attribute 'hide'}
	stRtDisableSetPos					: ST_CommandReturn;
	moveCCmdFB							: MC_PlanarFeedback;
	{attribute 'hide'}
	stRtMoveC							: ST_CommandReturn;
	adoptTrackOriCmdFB					: MC_PlanarFeedback;
	{attribute 'hide'}
	stRtAdoptTrackOri					: ST_CommandReturn;
	gearInPosOnTrackCmdFB				: MC_PlanarFeedbackGearInPosOnTrack;
	{attribute 'hide'}
	stRtGearInPosOnTrack				: ST_CommandReturnGearInPosOnTrack;
	gearInPosOnTrackMasterMoverCmdFB	: MC_PlanarFeedbackGearInPosOnTrackWithMasterMover;
	{attribute 'hide'}
	stRtGearInPosOnTrackMasterMover 	: ST_CommandReturnGearInPosOnTrackWithMasterMover;	
	setMoverPositionCmdFB 				: MC_PlanarFeedback;
	{attribute 'hide'}
	stRtSetMoverPosition				: ST_CommandReturn;
	
	// event logger
	aLog						: ARRAY[0..MAX_LAST_LOGS] OF ST_MoverCommandLog;
	{attribute 'hide'}
	fbResult					: FB_TcMoverMessage;		
	{attribute 'hide'}
	stTimeZoneInfo 				: TC2_UTILITIES.ST_TimeZoneInformation; //all times are UTC and must be converted to local time zone. if no timezone given only UTC times are avaialbe	
	{attribute 'hide'}
	_iErrID						: UDINT;
	{attribute 'hide'}
	_eLogSeverity				: TcEventSeverity := TcEventSeverity.VERBOSE;
	{attribute 'hide'}
	stLastCommand				: ST_MoverCommand;
	{attribute 'hide'}
	stActualMotionParameter		: ST_ActualMotionParameters;
	
	
	{attribute 'hide'}
	TrackTable					: ARRAY[0..maxTrackCount] OF ST_TrackTableInfo;
	{attribute 'hide'}
	nCycleCounter				: UDINT;	
	
	nLastKnownTrackOID			: OTCID;

	
END_VAR

{attribute 'hide'}
PROPERTY P_DcTimeStamp : ULINT
GET



P_DcTimeStamp := stMoverRef.MCTOPLC.SET.DcTimeStamp;
END_GET
END_PROPERTY

METHOD GetCommandLog : ST_MoverCommandLog
VAR_INPUT
	nNum	: UINT;
END_VAR
GetCommandLog := aLog[nNum];
END_METHOD

{attribute 'hide'}
METHOD MoverCommandToString : STRING
VAR_INPUT
	eMoverCommand : E_MoverCommandType;
END_VAR
CASE eMoverCommand OF
	eMoverCommand_eNoCommand :
		MoverCommandToString := 'eMoverCommand_eNoCommand';
	eMoverCommand_eMoveAbs :
		MoverCommandToString := 'eMoverCommand_eMoveAbs';
	eMoverCommand_eMoveModOnTrack : 
		MoverCommandToString := 'MoveOnTrack';
	eMoverCommand_eGearInPosOnTrack :
		MoverCommandToString := 'GearInPosOnTr';
	eMoverCommand_eGearInPosOnTrackMasterMover :
		MoverCommandToString := 'GInPoOnTrMMover';
	eMoverCommand_eMoveRel : 
		MoverCommandToString := 'eMoverCommand_eMoveRel';
	eMoverCommand_eHalt :
		MoverCommandToString := 'Halt'; 
	eMoverCommand_eHaltCa :
		MoverCommandToString := 'eMoverCommand_eHaltCa'; 					           
	eMoverCommand_eGearIn : 
		MoverCommandToString := 'eMoverCommand_eGearIn'; 				       
	eMoverCommand_eDynamicsChange : 
		MoverCommandToString := 'eMoverCommand_eDynamicsChange'; 		
	eMoverCommand_eGapChange : 
		MoverCommandToString := 'eMoverCommand_eGapChange'; 			   
	eMoverCommand_eSuperImposed : 
		MoverCommandToString := 'eMoverCommand_eSuperImposed'; 		   
	eMoverCommand_eCamInInstant : 
		MoverCommandToString := 'eMoverCommand_eCamInInstant'; 		   
	eMoverCommand_eCamInTwoTables : 
		MoverCommandToString := 'eMoverCommand_eCamInTwoTables'; 		
	eMoverCommand_eCamOut : 
		MoverCommandToString := 'eMoverCommand_eCamOut'; 				       
	eMoverCommand_eReset : 
		MoverCommandToString := 'Reset'; 				       
	eMoverCommand_eEnable : 
		MoverCommandToString := 'Enable';				       
	eMoverCommand_eDisable : 
		MoverCommandToString := 'Disable';				   
	eMoverCommand_eAddMoverToGroup: 
		MoverCommandToString := 'AddToGroup';		
	eMoverCommand_eRemoveMoverFromGroup : 
		MoverCommandToString := 'RemoveFromGroup';
	eMoverCommand_eMoveAbsDone :	
		MoverCommandToString := 'eMoverCommand_eMoveAbsDone';
    eMoverCommand_eMoveModDone :		
		MoverCommandToString := 'eMoverCommand_eMoveModDone';
    eMoverCommand_eMoveRelDone :		
		MoverCommandToString := 'eMoverCommand_eMoveRelDone';
	eMoverCommand_eHaltCaDone :		
		MoverCommandToString := 'eMoverCommand_eHaltCaDone';
    eMoverCommand_eMoveAbsQueueing :	
		MoverCommandToString := 'eMoverCommand_eMoveAbsQueueing';
    eMoverCommand_eMoveModQueueing :	
		MoverCommandToString := 'eMoverCommand_eMoveModQueueing';
    eMoverCommand_eMoveRelQueueing :	
		MoverCommandToString := 'eMoverCommand_eMoveRelQueueing';
    eMoverCommand_eGearInInSync :		
		MoverCommandToString := 'eMoverCommand_eGearInInSync';
    eMoverCommand_eGearOutOfSync :	
		MoverCommandToString := 'eMoverCommand_eGearOutOfSync';
	eMoverCommand_eMoveToPosition:	
		MoverCommandToString := 'MoveToPosition';
	eMoverCommand_eMoveToPositionXYC:	
		MoverCommandToString := 'MoveToPositionXYC';
	eMoverCommand_eMoveToPositionExt:	
		MoverCommandToString := 'MoveToPosExt';
	eMoverCommand_eJoinTrack:
		MoverCommandToString := 'Join Track';
	eMoverCommand_eLeaveTrack:
		MoverCommandToString := 'Leave Track';	
	eMoverCommand_eLeaveTrackInPosition:
		MoverCommandToString := 'Leave Track in Position';			
	eMoverCommand_eMoveZ:
		MoverCommandToString := 'Move Z';
	eMoverCommand_eMoveA:
		MoverCommandToString := 'Move A';
	eMoverCommand_eMoveB:	
		MoverCommandToString := 'Move B';
	eMoverCommand_eMoveC:	
		MoverCommandToString := 'Move C';
	eMoverCommand_eSetPosition:	
		MoverCommandToString := 'SetPos';		
	eMoverCommand_eEnableExternalSetPos:
		MoverCommandToString := 'En ExtSetGen';
	eMoverCommand_eDisableExternalSetPos :
		MoverCommandToString := 'Dis ExtSetGen';
		
		
		
		
	
END_CASE
END_METHOD

{attribute 'hide'}
METHOD UpdateCommandHistory
VAR_IN_OUT 
	stCommand : ST_MoverCommand;
END_VAR
VAR
	
END_VAR

VAR_INST
	lDCTime				: ULINT;
	fbTimeConvert 		: FB_FileTimeToTzSpecificLocalTime; 
	lTzCorrectDCTime 	: ULINT;
	stMoverAxisCommand 			: ST_MoverCommandLog; 
	stMoverAxisCommandClear 	: ST_MoverCommandLog; 
	fbFormatString		: FB_FormatString;
	nCntBuffer			: INT;
	TimeStampLength		: UDINT;
	corTimeStamp		: STRING;
	TimeStruct			: DCTIMESTRUCT;
	sDate				: STRING;
	sTime				: STRING;
	
	
	fTargetX			: LREAL;
	fTargetY			: LREAL;
	fTargetC			: LREAL;
	
	fbLoggerArgs	: FB_TcArguments;
	fbSourceInfo 	: FB_TcSourceInfo;
	

	
	tempString01	: T_MaxString;
	tempString02	: T_MaxString;
	tempString03	: T_MaxString;
	tempString04	: T_MaxString;
	tempString05	: T_MaxString;
	tempString06	: T_MaxString;
	tempString07	: T_MaxString;
	
END_VAR
	
	// Creating the timestamp
	lDCTime := F_GetActualDcTime64(); 
	fbTimeConvert(in:= DCTIME64_TO_FILETIME(lDcTime),tzInfo := stTimeZoneInfo); 
	lTzCorrectDCTime:= FILETIME_TO_DCTIME64(fbTimeConvert.out); 
	stCommand.stTimeStamp:= DCTIME64_TO_STRING( lTzCorrectDCTime); 
	corTimeStamp := DCTIME64_TO_STRING( lTzCorrectDCTime);
	stCommand.stTimeStamp := corTimeStamp;
	
	TimeStruct := DCTIME64_TO_DCTIMESTRUCT(lTzCorrectDCTime);
	
